// ---- DUTs/AxisControl/ST_AxisControlManualHMI.TcDUT
TYPE ST_AxisControlManualHMI :
STRUCT
	bEnableManualMode							: BOOL;
	bConsequentialError							: BOOL;
	bError										: BOOL;
	nErrorID									: UDINT;
	fSetPos										: LREAL;					// Set position (absolut value from NC)
	fModuloSetPos								: LREAL;					// Actual modulo position (absolut value from NC)
	fSetVelo									: LREAL;					// Set velocity
	fSetTorque									: LREAL;
	fActPos										: LREAL;					// Actual position (absolut value from NC)
	fModuloActPos								: LREAL;					// Actual modulo position (absolut value from NC)
	fActVelo									: LREAL;					// Actual velocity
	fActTorque									: LREAL;
	fPosDiff									: LREAL;					// Position difference (lag distance)
	stCommands									: ST_AxisControlManual;
	stStatus									: REFERENCE TO Tc2_MC2.ST_AxisStatus;
	stParameters								: REFERENCE TO Tc2_MC2.ST_AxisParameterSet;
END_STRUCT
END_TYPE

// ---- DUTs/CapPreScrewer/E_CapPreScrewer.TcDUT

(*
Nazwa:			E_GripperScrewerState
Opis:			Stan zakecarki szczekowej
Wersja:			v0.1
Data:			2023-10-10
Autor:			TW
Urzadzenia:		
Konfiguracja:	
Info:
*)

TYPE E_CapPreScrewer :
(	
	eReady							:= 10,
	ePreparingToPick				:= 20,			
	ePicking						:= 30,
	eVacumCheckPart1				:= 40,
	eVacumCheckPart2				:= 50,
	eVacumCheckPart3				:= 50,
	eVacumCheckPart4				:= 60,
	eTransferingVertical			:= 70,
	eTransferingHorizontal			:= 80,
	eAxisGearIn						:= 82,
	eVerticalDownToCatchPos			:= 90,
	ePositionOverBottle				:= 95,	
	eCatching						:= 100,		
	ePlacing						:= 110,
	eStrawCatcherBack				:= 120,
	eFinding						:= 130,
	eFindingStop					:= 140,
	ePreScrewing					:= 145,
	eScrewing						:= 150,
	eScrewingStop					:= 160,
	eFinished						:= 170,
	eGearOut						:= 175,
	                        		
	eReturning1						:= 180,
	eReturning2						:= 190,
                            		
			                	
	eDone							:= 200,
	eNotDone						:= 300
	


	
):= eReady;
END_TYPE

// ---- DUTs/CapPreScrewer/ST_ADS_Read_Write.TcDUT
TYPE ST_ADS_Read_Write :
STRUCT
	stCtr							: ST_ADS_Write;
	uiHardwerLimitSwitch			: UINT;
END_STRUCT
END_TYPE

// ---- DUTs/CapPreScrewer/ST_ADS_Write.TcDUT
TYPE ST_ADS_Write :
STRUCT
	uiNegativeTorqueLimit	AT %Q* : UINT := 2000;		//10 = 1%
	uiPositiveTorqueLimit	AT %Q* : UINT := 2000;
	siHardwerLimitSwitch		   : SINT;				//Hardwer limit switch: 0 - no limit switch, 1- NC, 1- NO
	
END_STRUCT
END_TYPE

// ---- DUTs/CapPreScrewer/ST_CapPreScrewerCommandsIn.TcDUT
TYPE ST_CapPreScrewerCommandsIn :
STRUCT
	bPendantDownwardMovement		: BOOL;						    // Kaseta sterownicza ruch do góry
	bPendantUpwardMovement			: BOOL; 						// Kaseta sterownicza ruch do dolu
	bPendantUpDownFast				: BOOL;							// Kaseta sterownicza góra/dól- wyższa prędkośc
	bPendantRightwardMovement		: BOOL; 						// Kaseta sterownicza ruch w prawo
	bPendantLeftwardMovement		: BOOL; 						// Kaseta sterownicza ruch w lewo
	bPendantRightLeftFast			: BOOL;							// Kaseta sterownicza lewo/prawo- wyższa prędkośc	
	bChoseRecipe					: BOOL;
	
END_STRUCT
END_TYPE

// ---- DUTs/CapPreScrewer/ST_CapPreScrewerParameters.TcDUT
TYPE ST_CapPreScrewerParameters :
STRUCT
	lrTopZPosition						: LREAL;		//Pozycja bezpieczna załapywarki na osi pionowej
	lrPickZPosition						: LREAL;		//Wysokość pobierania
	lrPickYPosition						: LREAL;		//Pozycja osi poziomej do pobierania
	lrPlaceZPosition					: LREAL;		//Wysokość odkładania - koniec załapywania gwintu
	lrPlaceYPosition					: LREAL;		//Pozycja osi poziomej do odkładania
	lrCartesianCatchZPosition			: LREAL;		//Wysokość osi Z dla zamykania łapacza słomek
	lrCapCatcherZPosition				: LREAL;		//Wysokość zamykaniałapek zakrętek
	lrStrawCatcherZPosition				: LREAL;		//Wysokość otwierania łapaczy słomek
	LrCheckStrawCatcherActuatorZPosition: LREAL;		//
	lrScrewerStartZPosition				: LREAL;		//Wysokość początku zakręcania
	lrGripperOpenPosition				: LREAL;		//Wysokość otwierania chwytaka szyjki butelki
	lrCapCapCatcherRelese				: LREAL;		//Wysokość otwierania chwytaka nakrętki
	lrCatcherTopPosition				: LREAL;		//Pozycja górna osi łapaczy słomek
	lrCatcherCatchingPosition			: LREAL;		//Pozycja łapania słomki
	lrCatcherPlacePosition				: LREAL;		//Pozycja dolna łapacza słomki
	lrCatcherSpeed						: LREAL;		//Prędkość 
	lrCatcherAcceleration				: LREAL;		//Przyspieszenie 
	lrCatcherJerk						: LREAL;		//Zryw 
	lrPickerSpeed						: LREAL;		//Prędkość 
	lrPickerSpeedWhenScrewer			: LREAL;		//Prędkość osi Z przy zakręcaniu
	lrPickerAcceleration				: LREAL;		//Przyspieszenie 
	lrPickerJerk						: LREAL;		//Zryw 
	lrScrewDistance						: LREAL;		//Kąt zakręcania
	lrScrewFinding						: LREAL;		//Kąt szukania gwintu
	lrScrewSpeed						: LREAL;		//Prędkość zakręcania
	lrScrewAcceleration					: LREAL;		//Przyspieszenie
	lrScrewJerk							: LREAL;		//Zryw
	lrBendingDistance					: LREAL;		//Odległość zaokrąglania ruchów manipulatora
	lrStrawInsertDistance				: LREAL;		//Odległość wspulnego ruchu osi Z i łapacza słomek (prowadzenie słomki) 
	
	lrCatcherMaxHight					: LREAL;		//Wysokość maksymalan łapacza słomek
	lrCatcherMinHight					: LREAL;		//Wysokość minimalan łapacza słomek
	lrCatcherHightSV					: LREAL;		//Nastawa wysokości łapacza słomek
	rCatcherHightOffset					: REAL;			//Pozycja bazowania
	rPulseRatio							: REAL;			//
	
	bPickerActiv						: ARRAY [1..4] OF BOOL;
	tTimeVacuumWatchdog					: TIME;

	lrHeightAdditionalBlow				: LREAL;		//Wysokość aktywacji dodatkowego przedmuchu wszystkich ssawek (od zakończenia nakładania nasadki)
	
	//bPicker2Activ						: BOOL;
	//bPicker3Activ						: BOOL;
	//bPicker4Activ						: BOOL;
	
	tWaitInPlacePos						: TIME;
	
	bStrawCatcherON						: BOOL;			//Aktywacja pracy łapacza słomek
	bRejectON							: BOOL;			//Aktywacja odrzucania nasadek przy nieudanym pobraniu
	bVacuumDeactivate					: BOOL;			//Deaktywować podcisnienie
	
	sADS_NetId							: STRING;		//Adres net id dla komunikacji ADS
	nAxisY_ADS_SlaveAddr				: UINT;			//Adres urzadzenia dla komunikacji ADS
	nAxisZ_ADS_SlaveAddr				: UINT;			//Adres urzadzenia dla komunikacji ADS
	nCatcher_ADS_SlaveAddr				: UINT;			//Adres urzadzenia dla komunikacji ADS
	
	lrBottleHight						: LREAL;		//Wysokość butelki
	lrCapHight							: LREAL;		//Wysokość zamknięcia
	lrCapNeckHight						: LREAL;		//Wysokość szyjki zamknięcia
	
END_STRUCT
END_TYPE

// ---- DUTs/CapPreScrewer/ST_FormsCapSorter.TcDUT
TYPE ST_FormsCapSorter :
STRUCT
	bFormPresence 			: BOOL;
	bBottlePresence			: BOOL;
	bFormControlCheck		: BOOL;
	bCapPutDown				: BOOL;
END_STRUCT
END_TYPE

// ---- DUTs/DUTsAdsCommunication/ST_Communication.TcDUT
TYPE ST_Communication :
STRUCT
	
	ePackMLMode						: Tc3_PackML.E_PMLUnitMode;						//Mode 
	ePackMLAutoState				: Tc3_PackML.E_PMLState;							//PackML Auto State
	sPackMLCommand					: ST_PackMLCmdForCom;					//PackML Commands
	
	eError							: S_Error;
	
	bEnable							: BOOL;	
	bCycleStart						: BOOL;
	bCycleStop						: BOOL;
	bCycleReset						: BOOL;
	bManualMode						: BOOL;
	bHoming							: BOOL;
	bHomingDone						: BOOL;	
	bConfectionEnding				: BOOL;
	tCycleTime						: TIME;
	iWatchdog						: INT;
	
	sRecipeName						: STRING(255);							
	sRecipeIndex					: STRING(255);
	
	eMachinePermissions				: ST_MachinePermissions;
	eReservedSignals				: ST_ReservedSignals;
END_STRUCT
END_TYPE

// ---- DUTs/DUTsAdsCommunication/ST_MachinePermissions.TcDUT
TYPE ST_MachinePermissions :
STRUCT
	(* REZERWA *)
	bPermission00 : BOOL;
	(* REZERWA *)
	bPermission01 : BOOL;
	(* REZERWA *)
	bPermission02 : BOOL;
	(* REZERWA *)
	bPermission03 : BOOL;
	(* REZERWA *)
	bPermission04 : BOOL;
	(* REZERWA *)
	bPermission05 : BOOL;
	(* REZERWA *)
	bPermission06 : BOOL;
	(* REZERWA *)
	bPermission07 : BOOL;
	(* REZERWA *)
	bPermission10 : BOOL;
	(* REZERWA *)
	bPermission11 : BOOL;
	(* REZERWA *)
	bPermission12 : BOOL;
	(* REZERWA *)
	bPermission13 : BOOL;
	(* REZERWA *)
	bPermission14 : BOOL;
	(* REZERWA *)
	bPermission15 : BOOL;
	(* REZERWA *)
	bPermission16 : BOOL;
	(* REZERWA *)
	bPermission17 : BOOL;
END_STRUCT
END_TYPE

// ---- DUTs/DUTsAdsCommunication/ST_PackMLCmdForCom.TcDUT
TYPE ST_PackMLCmdForCom :
STRUCT
	bStart						: BOOL;
	bHold						: BOOL;
	bUnHold						: BOOL;
	bSuspend					: BOOL;
	bAbort						: BOOL;
	bStop						: BOOL;
	bComplete					: BOOL;
	bClear						: BOOL;
	bReset						: BOOL;
	bStateComplete				: BOOL;	
END_STRUCT
END_TYPE

// ---- DUTs/DUTsAdsCommunication/ST_ReservedSignals.TcDUT
TYPE ST_ReservedSignals :
STRUCT
	(* REZERWA *)
	bReserved00 : BOOL;
	(* REZERWA *)
	bReserved01 : BOOL;
	(* REZERWA *)
	bReserved02 : BOOL;
	(* REZERWA *)
	bReserved03 : BOOL;
	(* REZERWA *)
	bReserved04 : BOOL;
	(* REZERWA *)
	bReserved05 : BOOL;
	(* REZERWA *)
	bReserved06 : BOOL;
	(* REZERWA *)
	bReserved07 : BOOL;
	(* REZERWA *)
	bReserved10 : BOOL;
	(* REZERWA *)
	bReserved11 : BOOL;
	(* REZERWA *)
	bReserved12 : BOOL;
	(* REZERWA *)
	bReserved13 : BOOL;
	(* REZERWA *)
	bReserved14 : BOOL;
	(* REZERWA *)
	bReserved15 : BOOL;
	(* REZERWA *)
	bReserved16 : BOOL;
	(* REZERWA *)
	bReserved17 : BOOL;
	(* REZERWA *)
	iReserved20 : INT;
	(* REZERWA *)
	iReserved30 : INT;
END_STRUCT
END_TYPE

// ---- DUTs/DUTsAxisOnline/FBsIO/ST_FBGetDriveRefIO.TcDUT
//==================================================================================================
//							Beckhoff Automation Poland
//									18.04.2018
//	Struktura zawierajaca I/O odpowiedniego bloku
//  v1.0	|| TC v 3.1.4022.16		|| - pierwsza wersja
//==================================================================================================
TYPE ST_FBGetDriveRefIO:
STRUCT
	bExecute						: BOOL;								// Rising edge executes cmd
	bBusy							: BOOL;								// Read/Write busy
	bError							: BOOL;								// Read/Write error
	udiErrorID						: UDINT;							// Read/Write error ID
END_STRUCT
END_TYPE

// ---- DUTs/DUTsAxisOnline/FBsIO/ST_FBHoldingBrakeCtrlIO.TcDUT
//==================================================================================================
//							Beckhoff Automation Poland
//									18.05.2018
//	Struktura zawierajaca I/O odpowiedniego bloku
//  v1.0	|| TC v 3.1.4022.16		|| - pierwsza wersja
//==================================================================================================
TYPE ST_FBHoldingBrakeCtrlIO:
STRUCT
	bForceLock 						: BOOL;								// 
	bForceUnlock					: BOOL;								// 
	bBusy							: BOOL;
	bError							: BOOL; 							// General error: parameter or CoE read.
																		// If bError = TRUE and bInitialized = FALSE - error during read motor data.
																		// If bError = TRUE and bInitialized = TRUE and (iAdsErrId <> 0 or iCANopenErrId <> 0) then I2T read error
																		// If bError = TRUE and bInitialized = TRUE and iAdsErrId = 0 and iCANopenErrId = 0 then parameter error: rTorqueLimit outside permitted range rTorqueLimitLow..rTorqueLimitHigh or Empty stDriveRef
	uiAdsErrId						: UINT;								// Forwarded output FB_CoERead_ByDriveRef
	uiSecErrId						: UINT;								// Sercos Error ID for AX5000, CanOpen error ID for AX8000
END_STRUCT
END_TYPE

// ---- DUTs/DUTsAxisOnline/FBsIO/ST_FBMotorMonitoringIO.TcDUT
//==================================================================================================
//							Beckhoff Automation Poland
//									21.05.2018
//	Struktura zawierajaca I/O odpowiedniego bloku
//  v1.0	|| TC v 3.1.4022.16		|| - pierwsza wersja
//==================================================================================================
TYPE ST_FBMotorMonitoringIO:
STRUCT
	bReset							: BOOL;								// Reset FB
	rTorqueLimit					: REAL		:=	500; 				// Bipolar torque limit: 0-500%, resolution 0.1%, value goes to: 16#6072 (Ch A)/ 16#6872 (Ch B)

	bError							: BOOL; 							// General error: parameter or CoE read.
																		// If bError = TRUE and bInitialized = FALSE - error during read motor data.
																		// If bError = TRUE and bInitialized = TRUE and (iAdsErrId <> 0 or iCANopenErrId <> 0) then I2T read error
																		// If bError = TRUE and bInitialized = TRUE and iAdsErrId = 0 and iCANopenErrId = 0 then parameter error: rTorqueLimit outside permitted range rTorqueLimitLow..rTorqueLimitHigh or Empty stDriveRef
	uiAdsErrId						: UINT;								// Forwarded output FB_CoERead_ByDriveRef
	uiSecErrId						: UINT;								// Sercos Error ID for AX5000, CanOpen error ID for AX8000
	bInitialized					: BOOL;								// TRUE - Motor data read without errors, so it's possible to calculate torqe and current values in metric units
	bWarning						: BOOL;								// rCurrentF > rWarningCurrent, be aware to be over permitted range
	rWarningCurrent					: REAL; 							// Continuous Stall Current - motor parameter: 16#6075 (Ch A)/ 16#6875 (Ch B); scalled: [A]
	rTorquePerc						: REAL;								// [%]
	rTorquePercMax					: REAL;								// Max [%]
	rTorque							: REAL; 							// [Nm]
	rTorqueF						: REAL;								// Filtered [Nm]
	rTorqueMax						: REAL;								// Max [Nm]
	rCurrent						: REAL; 							// [A]
	rCurrentF						: REAL;								// Filtered [A]
	rCurrentMax						: REAL;								// Max [A]
	rI2T							: REAL; 							// Thermal Motor Utilization: 16#32C1:02 (Ch A)/ 16#36C1:02 (Ch B); units: [%]
	rI2TMax							: REAL; 							// Max % Nominal
END_STRUCT
END_TYPE

// ---- DUTs/DUTsAxisOnline/FBsIO/ST_FBNcSWLimitSwitchCtrlIO.TcDUT
//==================================================================================================
//							Beckhoff Automation Poland
//									18.04.2018
//	Struktura zawierajaca I/O odpowiedniego bloku
//  v1.0	|| TC v 3.1.4022.16		|| - pierwsza wersja
//==================================================================================================
TYPE ST_FBNcSWLimitSwitchCtrlIO:
STRUCT
	bRead							: BOOL;								// Read SW limit switches values and states
	bWrite							: BOOL;								// Write SW limit switches values and states
	bReset							: BOOL; 							// Not yet
// Set values
	lrSetMinPos						: LREAL;							// SW limit switch minimum
	lrSetMaxPos						: LREAL;							// SW limit switch maximum
	bSetMinMon						: BOOL;								// Enable SW limit switch minimum monitoring
	bSetMaxMon						: BOOL;								// Enable SW limit switch maximum monitoring
// Actual values	
	lrActMinPos						: LREAL;							// Actual SW limit switch minimum
	lrActMaxPos						: LREAL;							// Actual SW limit switch maximum
	bActMinMon						: BOOL;								// SW limit switch minimum monitoring state
	bActMaxMon						: BOOL;								// SW limit switch maximum monitoring stateEND_STRUCT
//	
	bBusy							: BOOL;								// Read/Write busy
	bError							: BOOL;								// Read/Write error
	udiErrorID						: UDINT;							// Read/Write error ID
END_STRUCT
END_TYPE

// ---- DUTs/DUTsAxisOnline/FBsIO/ST_FBReadChannelErrorCodeIO.TcDUT
//==================================================================================================
//							Beckhoff Automation Poland
//									18.04.2018
//	Struktura zawierajaca I/O odpowiedniego bloku
//  v1.0	|| TC v 3.1.4022.16		|| - pierwsza wersja
//==================================================================================================
TYPE ST_FBReadChannelErrorCodeIO:
STRUCT
	bExecute						: BOOL;								// Rising edge executes cmd
	bBusy							: BOOL;
	bError							: BOOL; 							// General error: parameter or CoE read.
	uiAdsErrId						: UINT;								// Forwarded output FB_CoERead_ByDriveRef
	uiSecErrId						: UINT;								// Sercos Error ID for AX5000, CanOpen error ID for AX8000
	uiChannelErrorCode				: UINT;								// 603F Error code	0x603F (Ch A)/ 0x683F (Ch B) 	UINT16
	{attribute 'displaymode':='hex'}
	uiChannelErrorCodeHex			: UINT;								// 603F Error code	0x603F (Ch A)/ 0x683F (Ch B) 	UINT16
END_STRUCT
END_TYPE

// ---- DUTs/DUTsAxisOnline/FBsIO/ST_FBSetPositionOffsetIO.TcDUT
//==================================================================================================
//							Beckhoff Automation Poland
//									23.05.2018
//	Struktura zawierajaca I/O odpowiedniego bloku
//  v1.1	|| TC v 3.1.4022.16		|| - zmiana nazwy struktury usuniete CoE
//  v1.0	|| TC v 3.1.4022.16		|| - pierwsza wersja
//==================================================================================================
TYPE ST_FBSetPositionOffsetIO:
STRUCT
	bExecute						: BOOL;								// Rising edge executes cmd
	lrPosition						: LREAL;
	bRelative						: BOOL;
	eFeedback						: Tc2_MC2_Drive.E_PositionOffsetFeedback;
	eMemory							: Tc2_MC2_Drive.E_PositionOffsetMemory;
	bBusy							: BOOL;
	bError							: BOOL;
	udiErrorID						: UDINT;
	uiSecErrId						: UINT;								// Sercos Error ID for AX5000, CanOpen error ID for AX8000
END_STRUCT
END_TYPE

// ---- DUTs/DUTsAxisOnline/FBsIO/ST_McAxisOnlineErrorCollection.TcDUT
//==================================================================================================
//							Beckhoff Automation Poland
//									7.12.2018
//	Struktura zawierajaca wszsytkie bbledy AxisOnline
//  v1.1	|| TC v 3.1.4022.27		|| - dodane opisy bledow w formie zmiennych typu string
//  v1.0	|| TC v 3.1.4022.16		|| - pierwsza wersja
//==================================================================================================
TYPE ST_McAxisOnlineErrorCollection :
STRUCT
	// Error Collection
	bError							: BOOL;						// General Error flag - all error, FB, NC, drive, communication...
	bNcError						: BOOL;
	bFBError						: BOOL;						// Mc FB error
	bCommunicationError				: BOOL;						// ADS, CoE (AX8000), SoE (AX5000)...
	bDriveError						: BOOL;
	uiAdsErrorID					: UINT;						// Forwarded output FB_CoERead_ByDriveRef
	uiSecErrorID					: UINT;						// Sercos Error ID for AX5000, CanOpen error ID for AX8000
	udiErrorID						: UDINT;					// Set Position Offset FB error ID
	udiNcErrorID					: UDINT;					// Nc ErrorID
	{attribute 'displaymode':='hex'}
	udiNcErrorIDHex					: UDINT;					// Nc ErrorID
	udiFBErrorID					: UDINT;					// FB ErrorID
	{attribute 'displaymode':='hex'}
	udiFBErrorIDHex					: UDINT;					// FB ErrorID

	uiDriveErrorID					: UINT;						// 603F Error code	0x603F (Ch A)/ 0x683F (Ch B) 	UINT16
	{attribute 'displaymode':='hex'}
	uiDriveErrorIDHex				: UINT;						// 603F Error code	0x603F (Ch A)/ 0x683F (Ch B) 	UINT16
	sNcError						: STRING(255);				// Error description
	sDriveError						: STRING(255);				// Error description
END_STRUCT
END_TYPE

// ---- DUTs/DUTsAxisOnline/FBsIO/ST_McAxisStatus.TcDUT
//==================================================================================================
//							Beckhoff Automation Poland
//									24.04.2018
//	Struktura zawierajaca najwazniejsze statusy osi
//  v1.0	|| TC v 3.1.4022.16		|| - pierwsza wersja
//==================================================================================================
TYPE ST_McAxisStatus :
STRUCT
	stAxisStatus			: Tc2_MC2.ST_AxisStatus;
	sAxisName				: STRING(31);				// 
	dwAxisId				: DWORD;					// Axis ID
	bNcError				: BOOL;						// Nc Eror flag
	udiNcErrorCode			: UDINT;					// Nc axis error code
	{attribute 'displaymode':='hex'}
	udiNcErrorCodeHex		: UDINT;					// Nc axis error code - hex format
	lrActPos				: LREAL;					// Actual position (absolut value from NC)
	lrModuloActPos			: LREAL;					// Actual modulo position (absolut value from NC)
	lrActVelo				: LREAL;					// Actual velocity
	lrActAcc				: LREAL;					// Actual acceleration
	lrActTorque				: LREAL;
	lrSetPos				: LREAL;					// Set position (absolut value from NC)
	lrSetVelo				: LREAL;					// Set velocity
	lrSetAcc				: LREAL;					// Set acceleration
	lrSetTorque				: LREAL;

	lrPosDiff				: LREAL;					// Position difference (lag distance)
	bAxisReady				: BOOL;						// Axis.Status.Operational
	bHomed					: BOOL;
	bCoupled				: BOOL;
	bAcceptBlockedDrive		: BOOL;						// Force move back from limit switch
END_STRUCT
END_TYPE

// ---- DUTs/DUTsAxisOnline/FBsIO/ST_MCHaltIO.TcDUT
//==================================================================================================
//							Beckhoff Automation Poland
//									18.04.2018
//	Struktura zawierajaca I/O odpowiedniego bloku
//  v1.0	|| TC v 3.1.4022.16		|| - pierwsza wersja
//==================================================================================================
TYPE ST_MCHaltIO:
STRUCT
	bExecute						: BOOL;								// Rising edge executes cmd
	lrDeceleration					: LREAL;
	lrJerk							: LREAL;
	eBufferMode						: Tc2_MC2.MC_BufferMode;
	stOptions						: Tc2_MC2.ST_MoveOptions;
	bDone							: BOOL;
	bBusy							: BOOL;
	bActive							: BOOL;
	bCommandAborted					: BOOL;
	bError							: BOOL;
	udiErrorID						: UDINT;
END_STRUCT
END_TYPE

// ---- DUTs/DUTsAxisOnline/FBsIO/ST_MCHomeIO.TcDUT
//==================================================================================================
//							Beckhoff Automation Poland
//									18.04.2018
//	Struktura zawierajaca I/O odpowiedniego bloku
//  v1.0	|| TC v 3.1.4022.16		|| - pierwsza wersja
//==================================================================================================
TYPE ST_MCHomeIO:
STRUCT
	bExecute						: BOOL;								// Rising edge executes cmd
	lrPosition						: LREAL					:= DEFAULT_HOME_POSITION;
	eHomingMode						: Tc2_MC2.MC_HomingMode;
	eBufferMode						: Tc2_MC2.MC_BufferMode;
	stOptions						: Tc2_MC2.ST_HomingOptions;
	bCalibrationCam					: BOOL;
	bDone							: BOOL;
	bBusy							: BOOL;
	bActive							: BOOL;
	bCommandAborted					: BOOL;
	bError							: BOOL;
	udiErrorID						: UDINT;
END_STRUCT
END_TYPE

// ---- DUTs/DUTsAxisOnline/FBsIO/ST_MCJogIO.TcDUT
//==================================================================================================
//							Beckhoff Automation Poland
//									18.04.2018
//	Struktura zawierajaca I/O odpowiedniego bloku
//  v1.0	|| TC v 3.1.4022.16		|| - pierwsza wersja
//==================================================================================================
TYPE ST_MCJogIO:
STRUCT
	bSlowForward					: BOOL;
	bSlowBackward					: BOOL;
	bFastForward					: BOOL;
	bFastBackward					: BOOL;
	bJogForward						: BOOL;
	bJogBackwards					: BOOL;
	eMode							: Tc2_MC2.E_JogMode;
	lrPosition						: LREAL;
	lrVelocity						: LREAL;
	lrAcceleration					: LREAL;
	lrDeceleration					: LREAL;
	lrJerk							: LREAL;
	bDone							: BOOL;
	bBusy							: BOOL;
	bActive							: BOOL;
	bCommandAborted					: BOOL;
	bError							: BOOL;
	udiErrorID						: UDINT;
END_STRUCT
END_TYPE

// ---- DUTs/DUTsAxisOnline/FBsIO/ST_MCMoveAbsoluteIO.TcDUT
//==================================================================================================
//							Beckhoff Automation Poland
//									18.04.2018
//	Struktura zawierajaca I/O odpowiedniego bloku
//  v1.0	|| TC v 3.1.4022.16		|| - pierwsza wersja
//==================================================================================================
TYPE ST_MCMoveAbsoluteIO:
STRUCT
	bExecute						: BOOL;								// Rising edge executes cmd
	lrPosition						: LREAL;
	lrVelocity						: LREAL;
	lrAcceleration					: LREAL;
	lrDeceleration					: LREAL;
	lrJerk							: LREAL;
	eBufferMode						: Tc2_MC2.MC_BufferMode;
	stOptions						: Tc2_MC2.ST_MoveOptions;
	bDone							: BOOL;
	bBusy							: BOOL;
	bActive							: BOOL;
	bCommandAborted					: BOOL;
	bError							: BOOL;
	udiErrorID						: UDINT;
END_STRUCT
END_TYPE

// ---- DUTs/DUTsAxisOnline/FBsIO/ST_MCMoveModuloIO.TcDUT
//==================================================================================================
//							Beckhoff Automation Poland
//									18.04.2018
//	Struktura zawierajaca I/O odpowiedniego bloku
//  v1.0	|| TC v 3.1.4022.16		|| - pierwsza wersja
//==================================================================================================
TYPE ST_MCMoveModuloIO:
STRUCT
	bExecute						: BOOL;								// Rising edge executes cmd
	lrPosition						: LREAL;
	lrVelocity						: LREAL;
	lrAcceleration					: LREAL;
	lrDeceleration					: LREAL;
	lrJerk							: LREAL;
	eDirection						: Tc2_MC2.MC_Direction 		:= MC_Positive_Direction; // MC_Positive_Direction := 1, MC_Shortest_Way, MC_Negative_Direction, MC_Current_Direction
	eBufferMode						: Tc2_MC2.MC_BufferMode;
	stOptions						: Tc2_MC2.ST_MoveOptions;
	bDone							: BOOL;
	bBusy							: BOOL;
	bActive							: BOOL;
	bCommandAborted					: BOOL;
	bError							: BOOL;
	udiErrorID						: UDINT;
END_STRUCT
END_TYPE

// ---- DUTs/DUTsAxisOnline/FBsIO/ST_MCMoveRelativeIO.TcDUT
//==================================================================================================
//							Beckhoff Automation Poland
//									18.04.2018
//	Struktura zawierajaca I/O odpowiedniego bloku
//  v1.0	|| TC v 3.1.4022.16		|| - pierwsza wersja
//==================================================================================================
TYPE ST_MCMoveRelativeIO:
STRUCT
	bExecute						: BOOL;								// Rising edge executes cmd
	lrDistance						: LREAL;
	lrVelocity						: LREAL;
	lrAcceleration					: LREAL;
	lrDeceleration					: LREAL;
	lrJerk							: LREAL;
	eBufferMode						: Tc2_MC2.MC_BufferMode;
	stOptions						: Tc2_MC2.ST_MoveOptions;
	bDone							: BOOL;
	bBusy							: BOOL;
	bActive							: BOOL;
	bCommandAborted					: BOOL;
	bError							: BOOL;
	udiErrorID						: UDINT;
END_STRUCT
END_TYPE

// ---- DUTs/DUTsAxisOnline/FBsIO/ST_MCMoveVelocityIO.TcDUT
//==================================================================================================
//							Beckhoff Automation Poland
//									18.04.2018
//	Struktura zawierajaca I/O odpowiedniego bloku
//  v1.0	|| TC v 3.1.4022.16		|| - pierwsza wersja
//==================================================================================================
TYPE ST_MCMoveVelocityIO:
STRUCT
	bExecute						: BOOL;								// Rising edge executes cmd
	lrVelocity						: LREAL;
	lrAcceleration					: LREAL;
	lrDeceleration					: LREAL;
	lrJerk							: LREAL;
	eDirection						: Tc2_MC2.MC_Direction 		:= MC_Positive_Direction; // MC_Positive_Direction := 1, MC_Shortest_Way, MC_Negative_Direction, MC_Current_Direction
	eBufferMode						: Tc2_MC2.MC_BufferMode;
	stOptions						: Tc2_MC2.ST_MoveOptions;
	bDone							: BOOL;
	bInVelocity						: BOOL;								// The same meaning as bDone
	bBusy							: BOOL;
	bActive							: BOOL;
	bCommandAborted					: BOOL;
	bError							: BOOL;
	udiErrorID						: UDINT;
END_STRUCT
END_TYPE

// ---- DUTs/DUTsAxisOnline/FBsIO/ST_MCPowerIO.TcDUT
//==================================================================================================
//							Beckhoff Automation Poland
//									18.04.2018
//	Struktura zawierajaca I/O odpowiedniego bloku
//  v1.0	|| TC v 3.1.4022.16		|| - pierwsza wersja
//==================================================================================================
TYPE ST_MCPowerIO:
STRUCT
	bEnable							: BOOL;
	bEnable_Positive				: BOOL;
	bEnable_Negative				: BOOL;
	lrOverride						: LREAL := 100.0;
	eBufferMode						: Tc2_MC2.MC_BufferMode;
	stOptions						: Tc2_MC2.ST_PowerOptions;
	bStatus							: bool; // Same meaning as Done
	bBusy							: BOOL;
	bActive							: BOOL;
	bError							: BOOL;
	udiErrorID						: UDINT;
END_STRUCT
END_TYPE

// ---- DUTs/DUTsAxisOnline/FBsIO/ST_MCReadDriveAddressIO.TcDUT
//==================================================================================================
//							Beckhoff Automation Poland
//									18.04.2018
//	Struktura zawierajaca I/O odpowiedniego bloku
//  v1.0	|| TC v 3.1.4022.16		|| - pierwsza wersja
//==================================================================================================
TYPE ST_MCReadDriveAddressIO:
STRUCT
	bExecute						: BOOL;								// Rising edge executes cmd
	bDone							: BOOL;
	bBusy							: BOOL;
	bError							: BOOL;
	udiErrorID						: UDINT;
END_STRUCT
END_TYPE

// ---- DUTs/DUTsAxisOnline/FBsIO/ST_MCReadParameterSetIO.TcDUT
//==================================================================================================
//							Beckhoff Automation Poland
//									18.04.2018
//	Struktura zawierajaca I/O odpowiedniego bloku
//  v1.0	|| TC v 3.1.4022.16		|| - pierwsza wersja
//==================================================================================================
TYPE ST_MCReadParameterSetIO :
STRUCT
	bExecute						: BOOL;								// Rising edge executes cmd
	bDone							: BOOL;
	bBusy							: BOOL;
	bError							: BOOL;
	udiErrorID						: UDINT;
END_STRUCT
END_TYPE

// ---- DUTs/DUTsAxisOnline/FBsIO/ST_MCResetIO.TcDUT
//==================================================================================================
//							Beckhoff Automation Poland
//									18.04.2018
//	Struktura zawierajaca I/O odpowiedniego bloku
//  v1.0	|| TC v 3.1.4022.16		|| - pierwsza wersja
//==================================================================================================
TYPE ST_MCResetIO:
STRUCT
	bExecute						: BOOL;								// Rising edge executes cmd
	bDone							: BOOL;
	bBusy							: BOOL;
	bError							: BOOL;
	udiErrorID						: UDINT;
END_STRUCT
END_TYPE

// ---- DUTs/DUTsAxisOnline/FBsIO/ST_MCSetPositionIO.TcDUT
//==================================================================================================
//							Beckhoff Automation Poland
//									18.04.2018
//	Struktura zawierajaca I/O odpowiedniego bloku
//  v1.0	|| TC v 3.1.4022.16		|| - pierwsza wersja
//==================================================================================================
TYPE ST_MCSetPositionIO:
STRUCT
	bExecute						: BOOL;								// Rising edge executes cmd
	lrPosition						: LREAL;
	bMode							: BOOL;								// RELATIVE = True, ABSOLUTE = False (Default)
	stOptions						: Tc2_MC2.ST_SetPositionOptions;
	bDone							: BOOL;
	bBusy							: BOOL;
	bError							: BOOL;
	udiErrorID						: UDINT;
END_STRUCT
END_TYPE

// ---- DUTs/DUTsAxisOnline/FBsIO/ST_MCStopIO.TcDUT
//==================================================================================================
//							Beckhoff Automation Poland
//									18.04.2018
//	Struktura zawierajaca I/O odpowiedniego bloku
//  v1.0	|| TC v 3.1.4022.16		|| - pierwsza wersja
//==================================================================================================
TYPE ST_MCStopIO:
STRUCT
	bExecute						: BOOL;								// Rising edge executes cmd
	lrDeceleration					: LREAL; 
	lrJerk							: LREAL;
	stOptions						: Tc2_MC2.ST_MoveOptions;
	bDone							: BOOL;
	bBusy							: BOOL;
	bActive							: BOOL;
	bCommandAborted					: BOOL;
	bError							: BOOL;
	udiErrorID						: UDINT;
END_STRUCT
END_TYPE

// ---- DUTs/DUTsAxisOnline/ST_AX5000Diag.TcDUT
TYPE ST_AX5000Diag :
STRUCT
(* NC-Status *)
	nNCAxisID							: UDINT;
	bOperational						: BOOL;
	bC1DError							: BOOL;
	bWcStateError						: BOOL;
	bAxisError							: BOOL;
	iAxisErrorCode						: UDINT;

(* Drive Diag *)
	strDriveType						: STRING(19);
	strMotorType						: STRING(31);
	wDriveStatus						: WORD;
	wClass1Diag							: WORD;
	stClass1Diag						: ST_AX5000_C1D;
	stDriveStatus						: ST_AX5000DriveStatus;
	stEcSlaveStateBits					: ST_EcSlaveStateBits;
	stEcSlaveState						: ST_EcSlaveState;
	bPreopToSafeOpError					: BOOL;
	bSafeOpToOpError					: BOOL;
	stCPxInvParamList					: ST_SoE_CPxInvParamList;
	iDiagNumber							: UDINT;
	stDiagNumberList					: ST_SoE_DiagNumList;
	strDiagMessage						: STRING;
END_STRUCT
END_TYPE

// ---- DUTs/DUTsAxisOnline/ST_McAxisOnline.TcDUT
//==================================================================================================
//							Beckhoff Automation Poland
//									18.05.2018
//	Struktura interfejsu do obslugi Axis Online
//	v1.1	|| TC v 3.1.4022.16		|| - zmiana nazw struktur 
// 									 ST_FBCoEAX8000SetPositionOffsetIO 	--> ST_FBCoESetPositionOffsetIO
// 									 ST_FBHoldingBrakeCtrlAX8000IO 		--> ST_FBHoldingBrakeCtrlIO
// 									 ST_FBMotorMonitoringAX8000IO 		--> ST_FBMotorMonitoringIO
//  v1.0	|| TC v 3.1.4022.16		|| - pierwsza wersja
//==================================================================================================
TYPE ST_McAxisOnline :
STRUCT
	// Base administration
	mcPower							: ST_MCPowerIO;
	mcStop							: ST_MCStopIO;
	mcHalt							: ST_MCHaltIO;
	mcSS1							: ST_MCStopIO;
	mcSS2							: ST_MCStopIO;
	mcReset							: ST_MCResetIO;
	mcHome							: ST_MCHomeIO;
	mcSetPosition					: ST_MCSetPositionIO;
	stSetPositionOffset				: ST_FBSetPositionOffsetIO;
	// Base move
	mcMoveAbsolute					: ST_MCMoveAbsoluteIO;
	mcMoveRelative					: ST_MCMoveRelativeIO;
	mcMoveVelocity					: ST_MCMoveVelocityIO;
	mcMoveModulo					: ST_MCMoveModuloIO;
	mcMoveAbsolute2					: ST_MCMoveAbsoluteIO;
	mcMoveRelative2					: ST_MCMoveRelativeIO;
	mcMoveVelocity2					: ST_MCMoveVelocityIO;
	mcMoveModulo2					: ST_MCMoveModuloIO;
	mcJog							: ST_MCJogIO;
	// States, parameters, monitoring and diag
	stMotorMonitoring				: ST_FBMotorMonitoringIO;
	stHoldingBrake					: ST_FBHoldingBrakeCtrlIO;
	stNcLimitSwitch					: ST_FBNcSWLimitSwitchCtrlIO;
	stAxisParameter					: Tc2_MC2.ST_AxisParameterSet;
	stDriveRef						: Tc2_EtherCAT.ST_DriveRef;
	stDriveAddress					: Tc2_MC2.ST_DriveAddress;
	stChannelErrorCode				: ST_FBReadChannelErrorCodeIO;
	stStatus						: ST_McAxisStatus;
	// FBs
	stGetDriveRef					: ST_FBGetDriveRefIO;					// IO for FB_GetDriveRef
	mcReadDriveAddress				: ST_MCReadDriveAddressIO;				// IO for MC_ReadDriveAddress
	mcReadParameterSet				: ST_MCReadParameterSetIO;				// IO for MC_ReadParameterSet
	stError							: ST_McAxisOnlineErrorCollection;		// Error collection for all Axis Online functions
	bError							: BOOL;									// General Error flag - all error, FB, NC, drive, communication... check stError for detail
END_STRUCT
END_TYPE

// ---- DUTs/DUTsDiagnostics/E_DiagState.TcDUT
{attribute 'qualified_only'}
{attribute 'strict'}
TYPE E_DiagState :
(
	eOK						:= 10,
	eError					:= 20,
	eResetting				:= 30
);
END_TYPE

// ---- DUTs/DUTsDiagnostics/ST_FrmWcDiag.TcDUT
TYPE ST_FrmWcDiag :
STRUCT
	iNum					:DINT;
	sBin					:String;
END_STRUCT
END_TYPE

// ---- DUTs/DUTsNew/E_Actuator.TcDUT
{attribute 'qualified_only'}
{attribute 'strict'}
TYPE E_Actuator :
(
	eDisabled					:= 0,					// Stan nieaktywnosci             	
	eAborted                    := 1,                   // Stan bezpiecznego zatrzymania  
	eAborting                   := 2,                   // Stan bezpiecznego zatrzymywania
	eError                      := 3,                   // Stan bledu 				                                
	ePreparingToReady           := 7,                   // Stan przygotowywania do gotowosci           
	ePreparingToDisable         := 8,                   // Stan przygotowywania do nieaktywnosci                               
	eReady                      := 10,					// Stan gotowosci
	eResetting					:= 13,					// Stan resetowania bledu
	eRunningToPosition1			:= 15,       
	eRunningToPosition2			:= 16,                                          
	eRunning					:= 98,	                // Stan wykonywania ruchu 
    eNotdone                    := 99,	                // Stan niezakonczenia wykonywanego	                                     
    eDone                       := 100,                  // Stan zakonczenia wykonywanego ruchu   
	eDoneToPosition1            := 101,                  // Stan zakonczenia wykonywanego ruchu 
	eDoneToPosition2            := 102                  // Stan zakonczenia wykonywanego ruchu  
);
END_TYPE

// ---- DUTs/DUTsNew/E_Barrier.TcDUT
{attribute 'qualified_only'}
{attribute 'strict'}
TYPE E_Barrier :
(
	eDisabled 			:= 0,	
	eError				:= 1,				// Stan nieaktywnosci (Stacja wyłączona)             
	eReady				:= 2,				// Stan gotowści do ruchu
	eWaitingToClose		:= 20,				// Stan oczekiwania na zamknięcie ( 1 faza, 4 wagi)
	eWaitingToOpen		:= 21,				// Stan oczekiwania na otwaricie ( 1 faza, 2 wagi)
	eClose				:= 30,				// Stan zamykania
	eOpen				:= 40,				// Stan otwarcia
	eDone				:= 50				// Wykonano cykl 
):=eDisabled;
END_TYPE

// ---- DUTs/DUTsNew/E_WeightLiftStationState.TcDUT
TYPE E_WeightLiftStationState :
(
	eDisabled					:= 0,			//Stan wyłączony
	eReady						:= 10,			//Sprawdzam co się dzieje ze stacją
	ePrepareToStorageOfForms	:= 20,			//Przygotowywanie do magazynowania formatek
	eStorageOfForms				:= 30,			//Magazynuje formatki oraz podnoszę wagę
	eWeighingCycleStart			:= 40,			//Rozpoczęcie Ważenie
	eWeighingCycleON			:= 50,			//Ważenie
	eWeightLiftDown				:= 60,			//Opuszczanie formatek
	eDepartureOfForms			:= 70,			//Wypuszczamy formatki
	eDone						:= 80,			//Cykl skończony
	eRepair						:= 90			//Naprawa stacji
);
END_TYPE

// ---- DUTs/DUTsPackMLStateMachine/E_PackMLCommand.TcDUT
{attribute 'qualified_only'}
{attribute 'strict'}
TYPE E_PackMLCommand :
(
	eUndefined 				:= 0,
	eReset					:= 1,
	eStart					:= 2,
	eStop					:= 3,
	eHold					:= 4,
	eUnhold					:= 5,
	eSuspend 				:= 6,
	eUnsuspend				:= 7,
	eAbort 					:= 8,
	eClear					:= 9
	
);
END_TYPE

// ---- DUTs/DUTsPackMLStateMachine/E_PackMLMode.TcDUT
{attribute 'qualified_only'}
TYPE E_PackMLMode : 
(
	eUndefined		:=  0,
	eAutomatic		:=  1,
	eMaintenance 	:=  2,
	eManual 		:=  3
);
END_TYPE

// ---- DUTs/DUTsPackMLStateMachine/E_PackMLState.TcDUT
{attribute 'qualified_only'}
TYPE E_PackMLState : (
(* states according to PackTags v3.0 *)
	eUndefined				:=  0, //----Nieużywany
	eClearing 				:=  1, //----Nieużywany
	eStopped 				:=  2, //Błąd
	eStarting 				:=  3, //Uruchamianie
	eIdle 					:=  4, //Postój
	eSuspended 				:=  5, //---Nieużywany
	eExecute 				:=  6, //Praca
	eStopping	 			:=  7, //Zatrzymywanie
	eAborting 				:=  8, //Zatrzymywanie awaryjne
	eAborted 				:=  9, //Zatrzymano awaryjnie
	eHolding 				:= 10, //---Nieużywany
	eHeld 					:= 11, //---Nieużywany
	eUnholding 				:= 12, //---Nieużywany
	eSuspending 			:= 13, //---Nieużywany
	eUnsuspending 			:= 14, //---Nieużywany
	eResetting 				:= 15, //Resetowanie błędu, bazowanie
	eCompleting 			:= 16, //---Nieużywany
	eComplete	 			:= 17  //---Nieużywany
);
END_TYPE

// ---- DUTs/E_BottleFeederState.TcDUT
(*
Nazwa:			E_BottleFeederState
Opis:			Stan podajnika butlek
Wersja:			v0.1
Data:			2022-04-11
Autor:			DJ
Urzadzenia:		
Konfiguracja:	
Info:
*)
TYPE E_BottleFeederState :
(
	eDisabled					:= 0,  			// Wyłączona
	eError						:= 1, 			// Błąd 
	eReady						:= 2,			// Gotowość
	Homing						:= 3,    		// Bazowanie stacji 
	eHomingDone					:= 4,			// Bazowanie zakończone
	eManualMovements			:= 5,			// Tryb ręczny 
	ePreparingToMove			:= 60,			// Przygotowanie do ruchu
	eCloseFirstGate				:= 70,			// Zamknięcie pierwszego szlabanu
	eMoveToCatch				:= 80,			// Ruch do pobrania
	eCloseGripper				:= 90,			// Zamknięcie chwytaka
	eOpenSecondGate				:= 100,			// Otwarcie drugiego szlabanu
	eGoAbove					:= 110,			// Ruch nad formatkę
	eCloseSecondGate			:= 120,			// Zamknięcie drugiego szlabanu i otwarcie pierwszego
	eCloseStoper				:= 130, 			// Uruchomienie docisku
	eInsterting					:= 140,			// Wkładanie butelki
	eOpenGripper				:= 150,			// Otwieranie chwytaka
	eBackToPosition				:= 160,			// Powrót do pozycji wyjściowej
	eRelaseStoper				:= 170			// Wypuszczanie formatki 
);

END_TYPE

// ---- DUTs/E_CapFeederState.TcDUT
(*
Nazwa:			E_CapFeederState
Opis:			Stany sortera nasadek
Wersja:			v0.1
Data:			2018-10-10
Autor:			DP
Urzadzenia:		
Konfiguracja:	
Info:
*)


TYPE E_CapFeederState :
(
	eDisabled:=0,  		//Wyłączona
	eError:=1,			//Błąd
	eManualMovement:=2, //Tryb serwisowy
	eHoming:=3,			//Bazowanie
	eHomingDone:=4, 	//Koniec bazowania
	eReady:=5,			//Gotowość
	eSleeveLowLevel:=6, //Praca, Niski poziom
	eSorting:=7,		//Praca
	eSleeveFull:=8,		//Zapełniona
	ePreparingToDisable:=10 (*NOWY*) //Przygotowanie do wyłączenia
):=eDisabled;
END_TYPE

// ---- DUTs/E_CapFeederState_1.TcDUT
(*
Nazwa:			E_CapFeederState
Opis:			Stany sortera nasadek
Wersja:			v0.1
Data:			2022-07-13
Autor:			DP
Urzadzenia:		
Konfiguracja:	
Info:
*)


TYPE E_CapFeederState_1 :
(
	eDisabled:=0,			//Wyłączony
	eReady:=1,				//Gotowość
	eSleeveLowLevel:=2, 	//Praca, Niski poziom
	eSorting:=3,			//Praca
	eSleeveFull:=4			//Zapełniona
):=eDisabled;
END_TYPE

// ---- DUTs/E_CapPushingState.TcDUT
(*
Nazwa:			E_LidSealingState
Opis:			Stan wbijania nasadek
Wersja:			v0.1
Data:			2018-10-10
Autor:			TW
Urzadzenia:		
Konfiguracja:	
Info:
*)

TYPE E_CapPushingState :
(               	
	eReady:=1,				//Gotowość
	ePushing:=2,			//Wbijanie
	eHolding:=3,			//Przytrzymywanie
	ePushed:=4,				//Wbito
	eGoingUp:=5			//Podnoszenie
);
END_TYPE

// ---- DUTs/E_CatchStationState.TcDUT
(*
Nazwa:			E_CatchStationState
Opis:			Stany chwytaka
Wersja:			v0.2
Data:			2018-10-18
Autor:			TW
Urzadzenia:		
Konfiguracja:	
Info:
-nowy stan
*)

TYPE E_CatchStationState :
(
	eDisabled:=0,  			//Wyłączona
	eError:=1,				//Błąd
	eManualMovement:=2,		//Tryb serwisowy
	eHoming:=4,				//Bazowanie
	eHomingDone:=5,			//Koniec bazowania
	eReady:=6,				//Gotowość
	eCatching:=7, 			//Chwytanie
	eCatched:=8,  			//Chwycono
	ePreparingToDisable:=9, (*NOWY*) //Przygotowanie do wyłączenia
	eNotCatched:=10       //NIe złapało
):=eDisabled;
END_TYPE

// ---- DUTs/E_CheckerState.TcDUT
(*
Nazwa:			E_CheckerState
Opis:			Stan sprawdzania butelek
Wersja:			v0.3
Data:			2023-05-30
Autor:			DP
Urzadzenia:		
Konfiguracja:	
Info:

*)

TYPE E_CheckerState :
(
	eDisabled:=0,			//Wyłączona
	eError:=1,				//Błąd
	eManualMovement:=2,		//Tryb serwisowy
	eHoming:=3,				//Bazowanie
	eHomingDone:=4,			//Koniec bazowania
	eReady:=5,				//Gotowość
	eFormPresent:=6, 		//Formatka
	eBottleOK:=7,	 		//Butelka OK
	eLidOK:=8,		 		//Platynka OK
	eLidNOK:=9,		 		//Platynka NOK	
	eCapOK:=10,		 		//Nasadka OK
	eCapNOK:=11,		 	//Nasadka NOK
	ePreparingToDisable:=12,//Przygotowanie do wyłączenia
	eChecking := 20
):=eDisabled;
END_TYPE

// ---- DUTs/E_ConveyorState.TcDUT
(*
Nazwa:			E_ConveyorState
Opis:			Stan taśmociągu
Wersja:			v0.1
Data:			2018-10-10
Autor:			DP
Urzadzenia:		
Konfiguracja:	
Info:
*)
(*
TYPE E_ConveyorState :
(
	eDisabled:=0,		//Wyłączony
	eError:=1,			//Błąd
	eManualMovement:=2, //Tryb serwisowy
	eHoming:=3,			//Bazowanie
	eHomingDone:=4,		//Koniec bazowania
	eReady:=5,			//Gotowość
	eStopping:=6,	 //Zatrzymywanie
	eStarting:=7, 	//Uruchamianie
	eWorking:=8	  	//Praca
):=eDisabled;
END_TYPE
*)
TYPE E_ConveyorState :
(
	eDisabled := 0,						// Stan nieaktywnosci (Stacja wyłączona)             
	eAborted := 1,                   	// Stan bezpiecznego zatrzymania (po Abortingu) 
	eAborting := 2,                  	// Stan bezpiecznego zatrzymywania (po EStopie)
	eError := 3,                  	 	// Stan błędu 		
	eResetting := 4,					// Stan resetowania bledu (po Errorze)		                
	eManualMovement := 5,     			// Stan ruchów manualnych         
	eHoming := 6,						// Stan bazowania 
	eHomingDone := 7,                   // Stan wykonania bazowania 
	ePreparingToReady := 8,             // Stan przygotowywania do gotowosci (zawsze przed Ready)           
	ePreparingToDisable := 9,           // Stan przygotowywania do nieaktywnosci (po wyłączeniu Enable)                               
	eReady	:= 10,						// Stan gotowosci 
	eStopping := 11,					// Stan zatrzymywania 
	eStarting := 12,                  	// Stan uruchamiania (po Ready)
	eWorking := 13	               		// Stan wykonywania cyklu (po Startingu), w tym stanie osobny 
):=eDisabled;
END_TYPE

// ---- DUTs/E_DispencerLifterState.TcDUT
(*
Nazwa:			E_DispencerState
Opis:			Stan dozowników
Wersja:			v0.1
Data:			2018-10-10
Autor:			TW
Urzadzenia:		
Konfiguracja:	
Info:
*)

TYPE E_DispencerLifterState :
(
	eDisabled:=0,		//Wyłączony
	eError:=1,			//Błąd
	eManualMovement:=2,	//Tryb serwisowy
	eHoming:=3,			//Bazowanie
	eHomingDone:=4,		//Koniec bazowania
	eReady:=5,			//Gotowość
	ePreparingToDose:=6, //Przygotowanie dozy
	eDosingPh1:=7,		 //1 faza dozowania
	eDosingPh2:=8,		 //2 faza dozowania
	eDosingPh3:=9,		 //3 faza dozowania
	eDosingDone:=10,	 //Dozowanie  zakonczone
	eSucking:=11,		 //Pobieranie masy
	eGoingUp:=12,		 //Podnoszenie
	eAborting:=13,		 //Przerywanie
	ePreparingToDisable:=14,//Wylączanie
	ePulling:=15,		//Przeciaganie
(**)eDoseSucking:=16,	// Podsysanie
(**)eDoseSuckingDone:=17 //Koniec podsysania
):=eDisabled;
END_TYPE

// ---- DUTs/E_DispencerState.TcDUT
(*
Nazwa:			E_DispencerState
Opis:			Stan dozowników
Wersja:			v0.1
Data:			2022-03-15
Autor:			DP
Urzadzenia:		
Konfiguracja:	
Info:
- dodane mycie CIP
*)

TYPE E_DispencerState :
(
	eDisabled:=0,		 	//Wyłączony
	eReady:=5,			 	//Gotowość
	ePreparingToDose:=6, 	//Przygotowanie dozy
	eDosingPh1:=7,		 	//1 faza dozowania
	eDosingPh2:=8,		 	//2 faza dozowania
	eDosingPh3:=9,		 	//3 faza dozowania
	eDosingDone:=10,	 	//Dozowanie  zakonczone
	eDoseSucking:=11,	 	//Podsysanie
	eDoseSuckingDone:=12, 	//Koniec podsysania	
	eSucking:=13,		 	//Pobieranie masy
	eGoingUp:=14,		 	//Podnoszenie
	eAborting:=15,		 	//Przerywanie
	ePreparingToDisable:=16,//Wylączanie
	ePulling:=17,			//Przeciaganie
	eCleaningPreparing:=18,	//Mycie | przejazd do pozycji górnej
	eCleaningReady:=19,		//Mycie | pozycja tłoka w górze
	eCleaning:=20,			//Mycie | w trakcie ruchu w dół
	eCleaningDone:=21		//Mycie | pozycja tłoka w dole
):=eDisabled;
END_TYPE

// ---- DUTs/E_DragStationState.TcDUT
(*
Nazwa:			E_DragStationState
Opis:			Stan stacji przeciągania
Wersja:			v0.1
Data:			2021-10-14
Autor:			DJ
Urzadzenia:		
Konfiguracja:	
Info:
*)


TYPE E_DragStationState :
(
	eDisabled					:= 0,  			// Wyłączona
	eReady						:= 2,			// Gotowość
	ePreparingToMove			:= 4,			// Przygotowanie do ruchu
	eLifting					:= 7, 			// Podnoszenie
	ePrepareToDrag				:= 8, 			// Przygotowanie do przeicagana
	eDraging					:= 9,			// Przeciaganie
	eDragingDone				:= 10,			// Kończenie przeciągania
	eEndingOfDrag				:= 11,			// koniec przeciągania, poprawka pozycji
	eEndingOfDragDone			:= 12,			// koniec poprawki
	eLowering					:= 13,			//Opuszczanie 
	eDraged						:= 14,  		//Powrót do bazy, przeciągnięte
	eDragedDone					:= 15
):=eDisabled;

END_TYPE

// ---- DUTs/E_DragStationStatePneum.TcDUT
(*
Nazwa:			E_DragStationState
Opis:			Stan stacji przeciągania pneumatyczengo
Wersja:			v0.2
Data:			2022-05-18
Autor:			DJ
Urzadzenia:		Przeciąganie butelek
Konfiguracja:	
Info:
*)


TYPE E_DragStationStatePneum :
(
	eDisabled					:= 0,  			//Wyłączona
	eReady						:= 2,				//Gotowość
	ePreparingToMove			:= 4,	//Przygotowanie do ruchu
	eLifting					:= 7, 			//Podnoszenie
	ePrepareToDrag				:= 8, 		//Przygotowanie do przeicagana
	eDraging					:= 9,			//Przeciaganie
	eDragingDone				:= 10,
	eEndingOfDrag				:= 11,
	eEndingOfDragDone			:= 12,
	eLowering					:= 13,			//Opuszczanie 
	eDraged						:= 14,  			//Powrót do bazy, przeciągnięte
	eDragedDone					:= 15
):=eDisabled;

END_TYPE

// ---- DUTs/E_EntranceGatesState.TcDUT
(*
Nazwa:			E_EntranceGatesState
Opis:			Stan szlabanów
Wersja:			v0.1
Data:			2018-10-10
Autor:			TW
Urzadzenia:		
Konfiguracja:	
Info:
*)

TYPE E_EntranceGatesState :
(
	eDisabled:=0,					//Wyłączona
	eError:=1,						//Błąd
	eManualMovement:=2,				//Tryb serwisowy
	eHoming:=4,						//Bazowanie
	eHomingDone:=5,					//Koniec bazownia
	eReady:=6,						//Gotowość
	eInsertingTwoForms:=8,			//Wjazd 2 
	eInsertingOneForm:=9,			//Wjazd 1
	eWaitingForRealeseCommand:=11, 	//Czekanie
	eRealeseTwoForms:=12,			//Wyjazd 2
	eRealeseOneForm:=13,			//Wyjazd 1
	eBlocking:=14,					//Blokowanie (**)
	ePulling:=15,					//Przeciąganie (**)
	ePullingDone:=16,				//Wykonano przeciąganie (**)
	ePreparingToReady:=17,			//Przygotowanie do gotowości
	ePreparingToDisable:=18,		//Pryzgotowanie do wyłączenia
	ePullingToMiddle:=19,			//Przeciąganie do środka (**)
	ePullingToMiddleDone:=20,		//Przeciągnięto do środka(**)
	eStayOpen:=21			//Pozstań otwarty
	
):=eDisabled;
END_TYPE

// ---- DUTs/E_FestoEmcsStState.TcDUT
{attribute 'qualified_only'}
{attribute 'strict'}
TYPE E_FestoEmcsStState :
(
	eUnhomed		:=	0,
	eHoming			:=	5,
	eHomingDone		:=	7,
	eUnknown		:=	10,
	eIn				:=	20,
	eOut			:=	30,
	eInter			:=	40,
	eMoveIn			:=	50,
	eSettingIn		:=	55,
	ePlsIn			:=	56,
	eMoveOut		:=	60,
	eSettingOut		:=	65,
	ePlsOut			:=	66,
	eMoveInter		:=	70,
	eSettingInter	:=	75,
	eError			:=	100,
	eResetting		:=	200,
	eEStop			:=	1000						
);
END_TYPE

// ---- DUTs/E_GripperScrewer.TcDUT
(*
Nazwa:			E_GripperScrewerState
Opis:			Stan zakecarki szczekowej
Wersja:			v0.1
Data:			2018-10-10
Autor:			TW
Urzadzenia:		
Konfiguracja:	
Info:
*)

TYPE E_GripperScrewer :
(	
	
	eReady				:= 1,
	eToPushingPosition	:= 2,
	eToScrewingPosition	:= 3,
	ePushed				:= 4,			
	eFindingScrew		:= 5,			
	eScrewing			:= 6,			
	eGoingUp			:= 7,			
	eDone				:= 8,
	eNotDone			:= 9,
	eHolding			:= 10
	
):= eReady;
END_TYPE

// ---- DUTs/E_MachineState.TcDUT
(*
Nazwa:			E_MachineState
Opis:			Stan masyzny
Wersja:			v0.1
Data:			2018-10-10
Autor:			TW,DP
Urzadzenia:		
Konfiguracja:	
Info:
*)

//{attribute 'strict'}
//{attribute 'qualified_only'}
TYPE E_MachineState :
(
	eOn := 0, //Właczono
	ePower := 1, //Zasilanie
	eIdle := 2,	//Inicjacja
	eWaitingForPositioning := 4, //Czekanie na bazowanie
	ePositioning := 5, //Bazowanie
	eReady := 6, //Gotowa
	eServiceMode := 7, //Tryb Serwisowy
	eEnginesOn := 8, //Silniki włączone
	eCycleStarting := 9, //Start cyklu
	eCycleOn := 10, //Praca
	eStopping := 11, //Zatrzymywanie
	eConfectionStart := 12, //Start konfekcji
	eConfectionEnd := 13, //Stop konfekcji
	eHardError := 20, //Bład safety
	eSoftError := 21, //Bład
	eAfterError := 22, //Przywracanie po błedzie
	eReset := 30 //Resetowanie
);
END_TYPE

// ---- DUTs/E_MassHeatingState.TcDUT
(*
Nazwa:			E_MassHeatingState
Opis:			Stan grzania masy
Wersja:			v0.1
Data:			2018-10-10
Autor:			DP
Urzadzenia:		
Konfiguracja:	
Info:
*)

TYPE E_MassHeatingState :
(
	eDisabled:=0,		//Wyłączona
	eHeating:=1,		//Grzanie
	eReady:=2,			//Gotowość
	eCooling:=3			//Chłodzenie
);
END_TYPE

// ---- DUTs/E_PuckInserterState.TcDUT
(*
Nazwa:			E_PuckInserterState
Opis:			Stan podajnika opakowań
Wersja:			v0.1
Data:			2025-02-06
Autor:			DP
Urzadzenia:		
Konfiguracja:	
Info:
*)
TYPE E_PuckInserterState :
(
	eDisabled					:= 0,  			// Wyłączona
	eError						:= 1, 			// Błąd 
	eReady						:= 2,			// Gotowość
	ePreparingToMove			:= 60,			// Przygotowanie do ruchu
	eTurning					:= 70,			// Obrót
	eTurningDone				:= 80,			// Koniec obrotu
	eGoAbove					:= 110,			// Ruch nad formatkę
	eCloseStoper				:= 130, 		// Uruchomienie docisku
	eInsterting					:= 140,			// Wkładanie butelki
	eBackToPosition				:= 160			// Powrót do pozycji wyjściowej

);

END_TYPE

// ---- DUTs/E_RobotMovState.TcDUT
(*
Nazwa:			E_RobotPickAndPlace
Opis:			Stan robota pick-place
Wersja:			v0.1
Data:			2018-10-10
Autor:			TW
Urzadzenia:		
Konfiguracja:	
Info:
*)
TYPE E_RobotMovState :
(
	
	eReadyPlace						:= 0,		// robot w pozycji gotowości
	ePicking						:= 1,  		// pobieranie 
	ePicked							:= 2,
	ePlacing						:= 3,
    ePlaced							:= 4,
	eRejecting						:= 5,
	eRejected 						:= 6,
	eMovingInkJetStartPositon		:= 7,
	eMovedInkJetStartPositon		:= 8,
	eMovingInkJetStopPositon		:= 9,
	eMovedInkJetStopPositon			:= 10,
	eAborting						:= 11,
	eReturnToReadyPlace				:= 12,
	ePickingAfterEStop				:= 13,
	eMovingWeightPosition			:= 14,
	eMovedWeightPosition			:= 15,
	eMovingAfterWeightPosition		:= 16,
	eMovedAfterWeightPosition		:= 17,
	eMovingRotatedToPlace			:= 18,
	eMovedRoatedToPlace				:= 19
	
);
END_TYPE

// ---- DUTs/E_RollerScrewer.TcDUT
(*
Nazwa:			E_RollerScrewerState
Opis:			Stan zakręcarki rolkowej
Wersja:			v0.1
Data:			2018-10-10
Autor:			DP
Urzadzenia:		
Konfiguracja:	
Info:
*)
TYPE E_RollerScrewer :
(
	eDisabled		:=0,			//Niegotowy
	eReady			:=1,			//Gotowość 
	ePushingCap		:=2,			//Wciskanie
	ePushed			:=4,			//Wciśnięto
	eFindingScrew	:=5,			//Szukanie gwintu
	eScrewing		:=6,			//Zakręcanie
	eGoingUp		:=7,			//Podnoszenie
	eDone			:=8,			//Zakręcono
	eNotDone		:=9,			//Przerywanie
	eHolding		:=10			//Przytrzymywanie

):=eDisabled;
END_TYPE

// ---- DUTs/E_Station.TcDUT
(*
Nazwa:			E_MassHeatingState
Opis:			Stan grzania masy
Wersja:			v0.1
Data:			2018-10-10
Autor:			DP
Urzadzenia:		
Konfiguracja:	
Info:
*)

TYPE E_Station :
(
	eDisabled := 0,						// Stan nieaktywnosci (Stacja wyłączona)             
	eAborted := 1,                   	// Stan bezpiecznego zatrzymania (po Abortingu) 
	eAborting := 2,                  	// Stan bezpiecznego zatrzymywania (po EStopie)
	eError := 3,                  	 	// Stan błędu 		
	eResetting := 4,					// Stan resetowania bledu (po Errorze)		                
	eManualMovement := 5,     			// Stan ruchów manualnych         
	eHoming := 6,						// Stan bazowania 
	eHomingDone := 7,                   // Stan wykonania bazowania 
	ePreparingToReady := 8,             // Stan przygotowywania do gotowosci (zawsze przed Ready)           
	ePreparingToDisable := 9,           // Stan przygotowywania do nieaktywnosci (po wyłączeniu Enable)                               
	eReady	:= 10,						// Stan gotowosci 
	eStopping := 11,					// Stan zatrzymywania 
	eStarting := 12,                  	// Stan uruchamiania (po Ready)
	eRunning := 13,	               		// Stan wykonywania cyklu (po Startingu), w tym stanie osobny 
	eDone	:= 14			// Zakończony cykl running
);
END_TYPE

// ---- DUTs/E_WeightState.TcDUT
(*
Nazwa:			E_WeightState
Opis:			Stan zakręcarki rolkowej
Wersja:			v0.1
Data:			2018-10-10
Autor:			TW
Urzadzenia:		
Konfiguracja:	
Info:
*)
TYPE E_WeightState :
(
	eDisabled:=0,		//Wyłączona
	eReady:=1,	  		//Gotowa
	eWeighting:=2,		//Ważenie
	eWeightingDone:=3	//Koniec ważenia
);
END_TYPE

// ---- DUTs/ServerClientENUMS/E_ConnectionSteps.TcDUT
TYPE E_ConnectionSteps :
(
	eCONNECTION_STATE_IDLE,
	eCONNECTION_STATE_CONNECT_START,
	eCONNECTION_STATE_CONNECT_WAIT,
	eCONNECTION_STATE_DATAEXCHANGE,
	eCONNECTION_STATE_CLOSE_START,
	eCONNECTION_STATE_CLOSE_WAIT,
	eCONNECTION_STATE_ERROR
);
END_TYPE

// ---- DUTs/ServerClientENUMS/E_ServerSteps.TcDUT
TYPE E_ServerSteps :
(
	eSERVER_STATE_IDLE,
	eSERVER_STATE_LISTENER_OPEN_START,
	eSERVER_STATE_LISTENER_OPEN_WAIT,
	eSERVER_STATE_REMOTE_CLIENTS_COMM,
	eSERVER_STATE_REMOTE_CLIENTS_CLOSE,
	eSERVER_STATE_LISTENER_CLOSE_START,
	eSERVER_STATE_LISTENER_CLOSE_WAIT,
	eSERVER_STATE_ERROR
);
END_TYPE

// ---- DUTs/Stations/LidFeeder/E_LidFeederState.TcDUT
(*
Nazwa:			E_LidFeederState
Opis:			Stan zpodajnika platynek
Wersja:			v0.2
Data:			2018-10-18
Autor:			TW
Urzadzenia:		
Konfiguracja:	
Info:
*)

TYPE E_LidFeederState :
(
	eDisabled:=0,	//Wyłączona
	eError:=1,		//Błąd
	eManualMovement:=2,	//Tryb serwisowy
	eHoming:=3,		//Bazowanie
	eHomingDone:=4,	//Koniec bazowania
	eHeaterNotReady:=5,	//Grzanie
	eReady:=6,		//Gotowość
	eSuckingLid:=7,	//Pobieranie
	ePuttingLid:=8,	//Przygotowanie do odlożenia
	ePuttingLid2:=9,	//Nakładanie ostatnie
	eHeating:=10,	//Zgrzewanie
	eLidPutted:=11,	//Odłożona
	eGoingUp:=12,	//Podnoszenie
	ePreparingToDisable:=13 (*NOWY*) //Przygotowanie do wyłączenia
(**)
):=eDisabled;
END_TYPE

// ---- DUTs/Stations/LidSealer/E_LidSealing.TcDUT
(*
Nazwa:			E_LidSealingState
Opis:			Stan zgrzewarki platynek
Wersja:			v0.1
Data:			2018-10-10
Autor:			TW
Urzadzenia:		
Konfiguracja:	
Info:
*)

TYPE E_LidSealing :
(
	eDisabled:=0,		// Wyłączona
	eHeaterNotReady:=1, // Grzanie
	eReady:=2,			// Gotowość
	eSealing:=3,		// Zgrzewanie
	eHeating:=4,		// Grzanie
	eLidSealed:=5,		// Zgrzano
	eGoingUp:=6			// Podnoszenie
):=eDisabled;
END_TYPE

// ---- DUTs/Stations/WickFeeder/E_WickFeederSorterState.TcDUT
(*
Nazwa:			E_CapFeederState
Opis:			Stany sortera nasadek
Wersja:			v0.1
Data:			2018-10-10
Autor:			DP
Urzadzenia:		
Konfiguracja:	
Info:
*)


TYPE E_WickFeederSorterState :
(
	eDisabled:=0,  		//Wyłączona
	eError:=1,			//Błąd
	eManualMovement:=2, //Tryb serwisowy
	eHoming:=3,			//Bazowanie
	eHomingDone:=4, 	//Koniec bazowania
	eReady:=5,			//Gotowość
	eSleeveLowLevel:=6, //Praca, Niski poziom
	eSorting:=7,		//Praca
	eSleeveFull:=8,		//Zapełniona
	ePreparingToDisable:=10 (*NOWY*) //Przygotowanie do wyłączenia
):=eDisabled;
END_TYPE

// ---- DUTs/Stations/WickFeeder/E_WickFeederState.TcDUT
(*
Nazwa:			E_LidFeederState
Opis:			Stan zpodajnika platynek
Wersja:			v0.2
Data:			2018-10-18
Autor:			TW
Urzadzenia:		
Konfiguracja:	
Info:
*)

TYPE E_WickFeederState :
(
	eDisabled:=0,	//Wyłączona
	eError:=1,		//Błąd
	eManualMovement:=2,	//Tryb serwisowy
	eHoming:=3,		//Bazowanie
	eHomingDone:=4,	//Koniec bazowania
	//eHeaterNotReady:=5,	//Grzanie
	eFilling:=5,  //Zapełnianie zasobników
	eReady:=6,		//Gotowość 
	eWickDepotReady:=7,	//Magazynek przed włożeniem
	ePuttingWick:=8,	//Przygotowanie do odlożenia
	//ePuttingLid2:=9,	//Nakładanie ostatnie
	//eHeating:=10,	//Zgrzewanie
	eWickPutted:=11,	//Odłożona
	eGoingUp:=12,	//Podnoszenie
	ePreparingToDisable:=13 (*NOWY*) //Przygotowanie do wyłączenia
(**)
):=eDisabled;
END_TYPE

// ---- DUTs/ST_MoverState.TcDUT
TYPE ST_MoverState :
STRUCT
	bInPlacePosition			: BOOL; 	//Wózek w pozycji wyjmowania zamknięć	
	bPlaceAllowed				: BOOL;		//Zezwolenie na pobranie nasadki
	bInPickPosition				: BOOL; 	//Wózek w pozycjach wkładania zamknięć
	bMovingInPickPos			: BOOL;		//Wózek przemieszcza się w pozycji Pick 
	bWaitingForGoToPickPosition	: BOOL;		//Wózek czeka na przejscie do pick w biezpiecznej pozycji 
	bSlot1InPlacePosition		: BOOL;		//Gniazdo 1 ustawione w pozycji wkładania zamknięć
	bSlot2InPlacePosition		: BOOL;		//Gniazdo 2 ustawione w pozycji wkładania zamknięć
	bSlot3InPlacePosition		: BOOL;		//Gniazdo 3 ustawione w pozycji wkładania zamknięć
	bSlot4InPlacePosition		: BOOL;		//Gniazdo 4 ustawione w pozycji wkładania zamknięć
	stSlotStatus				: ARRAY [1..4] OF ST_SlotStatus;		//Gniazdo zapełnione
	bEmpty						: BOOL;		//Pusty wózek
	bFull						: BOOL; 	//zapełniony wózek
	iSlotNo						: INT;		//Nr gniazda
END_STRUCT
END_TYPE

// ---- DUTs/ST_Point.TcDUT
TYPE ST_Point :
STRUCT
	x : INT;
	y : INT;
END_STRUCT
END_TYPE

// ---- DUTs/ST_Point_1.TcDUT
TYPE ST_Point_1 :
STRUCT
	x : DT;
	y : INT;
END_STRUCT
END_TYPE

// ---- DUTs/ST_SlotStatus.TcDUT
TYPE ST_SlotStatus :
	STRUCT
		bFilled			: BOOL;
		bCupPlaced		: BOOL;
		bTubePresent	: BOOL;
		diPlacedRetry	: DINT;
	END_STRUCT
END_TYPE

// ---- DUTs/S_CycleTimes.TcDUT
(*
Nazwa:			S_CycleTimes
Opis:			Struktura czasów cyklu
Wersja:			v0.1
Data:			2019-08-29
Autor:			DP
Urzadzenia:		
Konfiguracja:	
Info:
*)
TYPE S_CycleTimes :
STRUCT
	bName:STRING; 
	bEnable:BOOL;
	dTime:DINT;
END_STRUCT
END_TYPE

// ---- DUTs/S_Error.TcDUT
(*
Nazwa:			S_Error
Opis:			Struktura bledu
Wersja:			v0.2
Data:			2018-10-10
Autor:			TW
Urzadzenia:		
Konfiguracja:	
Info:
- dodano string2
*)
TYPE S_Error :
STRUCT
	bError				: BOOL; 
	udiStationID		: UDINT;
	sStationName		: STRING;
	nErrorCode			: UDINT;
	sErrorString		: STRING(200);
	sErrorString2		: STRING(200);
	bReset:BOOL;
END_STRUCT
END_TYPE

// ---- DUTs/S_Information.TcDUT
(*
Nazwa:			S_Error
Opis:			Struktura bledu
Wersja:			v0.2
Data:			2018-10-10
Autor:			TW
Urzadzenia:		
Konfiguracja:	
Info:
- dodano string2
*)
TYPE S_Information :
STRUCT 
	udiID				: UDINT;
	wsDescription		: WSTRING;
END_STRUCT
END_TYPE

// ---- DUTs/S_PackageState.TcDUT
(*
Nazwa:			S_PackageState 
Opis:			Struktura formatki
Wersja:			v0.1
Data:			2018-10-10
Autor:			DP
Urzadzenia:		
Konfiguracja:	
Info:
*)
TYPE S_PackageState :
STRUCT
	
	nID									:UDINT;							//Numer butelki
	nCardNumber							:ULINT; 						//Numer karty RFID
	bFormPresent						:BOOL;							//Potwierdzenie obecności formatki na wjeździe karuzeli
	bBottlePresent						:BOOL;							//Potwierdzenie obecności butelki na wjeździe karuzeli
	bDosingTwoPhases					:BOOL;							//Jeżeli wybrano dozowanie dwu fazowe
	nDispencerNr						:INT;							//Numer dozownika który wydozował masę 1-6
	nDispencerNrSecondPhase				:INT;							//Numer dozownika który wydozował masę w drugiej fazie
	tDispencingTime						:TIME;							//Czas dozowania
	tDispencingTimeSecondPhase			:TIME;							//Czas dozowania w drugiej fazie
	lrDoseVolumeSV						:LREAL;							//Zadana wartość dozowania [ml]
	lrDoseVolumeCV						:LREAL;							//Aktualna wydozowana ilość [ml]
	lrDoseVolumeSVSecondPhase			:LREAL;							//Zadana wartość dozowania [ml]
	lrDoseVolumeCVSecondPhase			:LREAL;							//Aktualna wydozowana ilość [ml]
	bDosed								:BOOL;							//Zakońcozno cykl dozowania
	bDoseAborted						:BOOL;							//Przerwano dozowanie
	bDosedSecondPhase					:BOOL;							//Zakońcozno cykl dozowania 2 faz
	bDoseAbortedSecondPhase				:BOOL;							//Przerwano dozowanie 2faz
//	bFormInWheel1						:BOOL;							//Potwierdzenie obecności formatki na 1 wjeździe karuzeli
	bWeighed							:BOOL;							//Zwarzono paczkę
	bWeightAborted						:BOOL;							//Przerwano ważenie
	lrWeightSV							:LREAL;							//Zadana wartość netto [g] 
	lrWeightCV							:LREAL;							//Aktualna wartość netto [g]
	lrWeightMeasuredCV					:LREAL;							//Aktualna wartość odczytana z wagi [g]
	lrMinWeightCV						:LREAL;							//Minimalna waga wartość netto [g]	
	lrMaxWeightCV						:LREAL;							//Maksymalna waga wartość netto [g]		
	lrWeightDif							:LREAL;							//Różnica pomiarów				
	bWeightOK							:BOOL;							//Waga zgodna z zakresem tolerancji
	bWeightTooLow						:BOOL;							//Waga za niska
	bWeightTooHigh						:BOOL;							//Waga za wysoka
	tWeightingTime						:TIME;							//Czas ważenia
	bLidPutted							:BOOL;							//Platynka położona 
	bLidPutAborted						:BOOL;							//Odkładanie platynki wycofane w trakcie odkładania
	tLidPuttingTime						:TIME;							//Czas odkładania platynki
	lrPreSealingTime					:LREAL;							//Czas zgrzewania wstępnego
	lrPreSealingTemp					:LREAL;							//Temperatura zgrzewania wstępnego
	bLidPuttedChecked					:BOOL;							//Platynka sprawdzona 
	bLidPuttedOK						:BOOL;							//Platynka sprawidłowo nałożona
	bLidSealed							:BOOL;							//Platynka zgrzana
	bLidSealingAborted					:BOOL;							//Zgrzanie platynki wycofane
	tLidSealingTime						:TIME;							//Czas zgrzewania platynki
	lrLidSealingTemp					:LREAL;							//Temperatura zgrzewania zasadniczego
	bROPPPutted							:BOOL;							//ROPP nasadka ok
	bROPPPuttedChecked					:BOOL;							//ROPP nasadka sprawdzona
	bROPPCapped							:BOOL;							//ROPP ok
	bROPPCappingAborted					:BOOL;							//ROPP nok
	tROPPCappingTime					:TIME;							//Czas ROPPowania
	bROPPCappingOK						:BOOL;							//ROPP nasadka ok za
	bROPPCappingChecked					:BOOL;							
	bCapSorterPutted					:BOOL;							//Nałozono nakrętke przez sorter
	bCapSorterPuttedAborted				:BOOL;							//Nałozono nakrętke przez sorter	
	tCapSorterPuttingTime				:TIME;							//Czas Nałozono nakrętke przez sorter		
	bCapPutted							:BOOL;							//Nałozono nakrętke
	bCapPuttedNOK						:BOOL;							//Nałozono nakrętke NOK
	bCapChecked							:BOOL;							//Nakrętka sprawdzona
	bCapOK								:BOOL;							//Nakrętka OK
//	bCapPushed							:BOOL;							//Wbito nasadke
//	bCapPushingAborted					:BOOL;							//Przerwano wbijanie
//	tCapPushingTime						:TIME;							//Czas wbijania nasadki
//	bFormInWheel2						:BOOL;							//Potwierdzenie obecności formatki na 2 wjeździe karuzeli
	bCapGripperScrewed					:BOOL;							//Nakrętka zakręcona
	bCapGripperScrewAborted				:BOOL;							//Wycofanie z zakręcania nakrętki
	tCapGripperScrewingTime				:TIME;							//Czas zakręcania
//	bCapRollerScrewed					:BOOL;							//Nakrętka zakręcona
//	bCapRollerScrewAborted				:BOOL;							//Wycofanie z zakręcania nakrętki
//	tCapRollerScrewingTime				:TIME;							//Czas zakręcania
	bCapCorrectPutted					:BOOL;							//Nałozono nakrętke
	bCapCorrectChecked					:BOOL;							//Nakrętka sprawdzona
	bCapCorrectNOK						:BOOL;							//Nakrętka NOT OK
	bCapCorrectCapOn					:BOOL;							//Nakrętka obecna
	
	bCapCorrectCheckCameraOK			:BOOL;							//Nakrętka orientacja OK
	bCapCorrectCheckCameraChecked		:BOOL;							//Nakrętka orientacja sprawdzono
	
	bBottleTransferedToExit				:BOOL;							//Butelka przeniesiona na transporter odrzuconych butelek
	bBottleTransferedToLabeler			:BOOL;							//Butelka przeniesiona na etykieciarkę
	
	bTested								: BOOL;
	bTested2							: BOOL;
	bTested3							: BOOL;
	bTested4							: BOOL;
END_STRUCT
END_TYPE

// ---- DUTs/S_RFIDCheck.TcDUT
(*
Nazwa:			S_RFIDCheck
Opis:			sprawdzanie RFID
Wersja:			v0.1
Data:			2024-12-03
Autor:			
Urzadzenia:		
Konfiguracja:	
Info:

*)
TYPE S_RFIDCheck :
STRUCT 
	iNumber				: INT;		//Numer RFID	
	iReaded1			: INT;		//Odczytano z czytnika nr 1
	iReaded2			: INT;		//Odczytano z czytnika nr 2
	iReaded3			: INT;		//Odczytano z czytnika nr 3
	iReaded4			: INT;		//Odczytano z czytnika nr 4
	iReaded5			: INT;		//Odczytano z czytnika nr 5
END_STRUCT
END_TYPE

// ---- DUTs/S_Warning.TcDUT
(*
Nazwa:			S_Warning 
Opis:			Struktura ostrzezen
Wersja:			v0.1
Data:			2018-10-10
Autor:			DP
Urzadzenia:		
Konfiguracja:	
Info:
*)
TYPE S_Warning :
STRUCT
	bWarning:BOOL; 
	bAcknowledge:BOOL;
	sDescription:STRING;
	udiWarningCode:UDINT;
END_STRUCT
END_TYPE

// ---- POUs/Recipes/NewRecipes/Components/ST_BoolParametr.TcDUT
TYPE ST_BoolParametr :
STRUCT
	bValue												:	BOOL;
	bOldValue											:	BOOL;
	bDefault											:	BOOL;
	wsInfoCaption										:	WSTRING(100);
	wsCaption1											:	WSTRING(50);
	wsCaption2											:	WSTRING(50);
	bUse2caption										:	BOOL;
END_STRUCT
END_TYPE

// ---- POUs/Recipes/NewRecipes/Components/ST_DiParametrr.TcDUT
TYPE ST_DiParametrr :
STRUCT
	diValue											:	DINT;
	diOldValue											:	DINT;
	diMinLimit											:	DINT;
	diMaxLimit											:	DINT;
	diDefault											:	DINT;
	diColor											:	DINT	:=	16#FFFFAF1C;	
	wsInfoCaption										:	WSTRING(100);	
	wsCaption1											:	WSTRING(50);
	wsCaption2											:	WSTRING(50);
	bUse2caption										:	BOOL;
	wsUnit												:	WSTRING;
END_STRUCT
END_TYPE

// ---- POUs/Recipes/NewRecipes/Components/ST_LrParametr.TcDUT
TYPE ST_LrParametr :
STRUCT
	lrValue												:	LREAL;
	lrOldValue											:	LREAL;
	lrMinLimit											:	LREAL;
	lrMaxLimit											:	LREAL;
	lrDefault											:	LREAL;
	wsInfoCaption										:	WSTRING(120);	
	wsCaption1											:	WSTRING;
	wsCaption2											:	WSTRING;
	udiColor											:	UDINT	:=	16#FFF0F0F0;	
	bUse2caption										:	BOOL;
	wsUnit												:	WSTRING;
END_STRUCT
END_TYPE

// ---- POUs/Recipes/NewRecipes/Components/ST_TextListParametr.TcDUT
TYPE ST_TextListParametr :
STRUCT
	aWStringTable : ARRAY [0..3] OF WSTRING := ["Butelka okrągła", "Butelka płaska", "Słoik", "Karton jednostkowy"];
	eArrayNumber										:	E_ProductType;
END_STRUCT
END_TYPE

// ---- POUs/Recipes/NewRecipes/Components/ST_UdiParametr.TcDUT
TYPE ST_UdiParametr :
STRUCT
	udiValue											:	UDINT;
	udiOldValue											:	UDINT;
	udiMinLimit											:	UDINT;
	udiMaxLimit											:	UDINT;
	udiDefault											:	UDINT;
	udiColor											:	UDINT	:=	16#FFFFAF1C;	
	wsInfoCaption										:	WSTRING(100);	
	wsCaption1											:	WSTRING(50);
	wsCaption2											:	WSTRING(50);
	bUse2caption										:	BOOL;
	wsUnit												:	WSTRING;
END_STRUCT
END_TYPE

// ---- POUs/Recipes/NewRecipes/E_MacroProductProcessRegister.TcDUT
{attribute 'qualified_only'}
{attribute 'strict'}
TYPE E_MacroProductProcessRegister :
(
	eUnknown									:=	0,
	
	eEmpting									:=	10,
	eEmpty			 							:= 	20,
	
	ePuttingIn		 							:= 	30,
	eFull										:=	40,
	eNotFull									:=	50
//	ePickingToWait								:=	60,
//	ePickedAndWaiting							:=	70	
);
END_TYPE

// ---- POUs/Recipes/NewRecipes/E_ProductType.TcDUT
{attribute 'qualified_only'}
//{attribute 'strict'}
TYPE E_ProductType :
(

	eRoundBottle	:= 	0,
	eFlatBottle 	:= 	1,
	eJar			:=	2,	
	eCarton			:=	3
);
END_TYPE

// ---- POUs/Recipes/NewRecipes/RecipeList/E_FileOpSteps.TcDUT
{attribute 'qualified_only'}
{attribute 'strict'}
TYPE E_FileOpSteps :
(
	eNop 					:=	0,
	eStartOpen				:=	10,
	eWaitOpen				:=	20,
	eStartOper				:=	30,
	eWaitOper				:=	40,
	eStartClose				:=	50,
	eWaitClose				:=	60
);
END_TYPE

// ---- POUs/Recipes/NewRecipes/RecipeParts/ST_BoxRobotRecipe.TcDUT
TYPE ST_BoxRobotRecipe :
STRUCT
	wsCaption											:	WSTRING;	//Nazwa stacji	

	stPickOffsetX									:	ST_LrParametr;	//	Offset poz pobierania x 1mm
	stPickOffsetY									:	ST_LrParametr;	//	Offset poz pobierania x 1mm
	stPickOffsetZ									:	ST_LrParametr;	//	Offset poz pobierania x 1mm
	stPickOffsetA									:	ST_LrParametr;	//	Offset poz pobierania x 1 stopeń
	stPickOffsetB									:	ST_LrParametr;	//	Offset poz pobierania x 1 stopeń
	stPickOffsetC									:	ST_LrParametr;	//	Offset poz pobierania x 1 stopeń
	                                                                      	
	stPickAccelecation								:	ST_UdiParametr;	//	Acc in % [1..100]
	stPickDecceleration								:	ST_UdiParametr;	//	Dec in % [1..100]
	stPickOverride									:	ST_UdiParametr;	//	Override in % [1..100]
	stPickColisionDetect							:	ST_UdiParametr; //	Col awoid in %[1..100]
	stPickGripperDelayTime							:	ST_UdiParametr;	//	Czas dojazdu   ms
	stSuckingTimeOn									:	ST_UdiParametr;	//	Czas posysania ms
	stSuckingTimeOff								:	ST_UdiParametr; //	Czas posysania ms
                                                                          	
	stPlaceOffsetX									:	ST_LrParametr;	//	Offset poz odkladania 2 x 1mm
	stPlaceOffsetY									:	ST_LrParametr;	//	Offset poz odkladania 2 x 1mm
	stPlaceOffsetZ									:	ST_LrParametr;	//	Offset poz odkladania 2 x 1mm
	stPlaceOffsetA									:	ST_LrParametr;	//	Offset poz odkladania 2 x 1 stopeń
	stPlaceOffsetB									:	ST_LrParametr;	//	Offset poz odkladania 2 x 1 stopeń
	stPlaceOffsetC									:	ST_LrParametr;	//	Offset poz odkladania 2 x 1 stopeń
                                                                          	
	stPlaceAccelecation								:	ST_UdiParametr;	//	Acc in % [1..100]
	stPlaceDecceleration							:	ST_UdiParametr;	//	Dec in % [1..100]
	stPlaceOverride									:	ST_UdiParametr;	//	Override in % [1..100]
	stPlaceColisionDetect							:	ST_UdiParametr; //	Col awoid in %[1..100]
	stRezerwa1										:	ST_UdiParametr;	//	
	stRezerwa2										:	ST_UdiParametr; //	
	stRezerwa3										:	ST_UdiParametr;	//	
	stGripperTimeClose								:	ST_UdiParametr;	//	Czas skłądania chwytaka
	stGripperTimeOpen								:	ST_UdiParametr;	//	Czas otwierania chwytaka
	                                                                      	
	stPickPreX										:	ST_LrParametr;	//	Odsuniecie przed pozycją pobierania w osi X      
	stPickPreY										:	ST_LrParametr;	//	Odsuniecie przed pozycją pobierania w osi Y      	
	stPickPreZ										:	ST_LrParametr;	//	Odsuniecie przed pozycją pobierania w osi Z      
	stPickAfterX									:	ST_LrParametr;  //	Odsuniecie po pobraniu w osi X                   
	stPickAfterY		                            :	ST_LrParametr;  //	Odsuniecie po pobraniu w osi Y                   
	stPickAfterZ		                            :	ST_LrParametr;  //	Odsuniecie po pobraniu w osi Z                   
	stPlacePreX										:	ST_LrParametr;  //	Odsuniecie przed pozycją odłożenia w osi X       
	stPlacePreY		                                :	ST_LrParametr;  //	Odsuniecie przed pozycją odłożenia w osi Y       
	stPlacePreZ		                                :	ST_LrParametr;  //	Odsuniecie przed pozycją odłożenia w osi Z       
	stPlaceAfterX		                            :	ST_LrParametr;  //	Odsuniecie po odłożenia w osi X                  
	stPlaceAfterY		                            :	ST_LrParametr;  //	Odsuniecie po odłożenia w osi Y                  
	stPlaceAfterZ		                            :	ST_LrParametr;  //	Odsuniecie po odłożenia w osi Z                  
	stBoxPickHeight									:	ST_LrParametr;       
	stBoxWingDown	  	                            :	ST_LrParametr;  //	Dolna długość krawędzi skrzydła kartonu          
	stCurveMotionPositionZ	  	                    :	ST_LrParametr;  //	Wysokość osłon dla dokładnego wkładania
	stCurveDistanceX	                            :	ST_LrParametr;  //	Offset pozycji najeżdzania na balchę prowadzącą X
	stCurveDistanceY								:	ST_LrParametr;  //	Offset pozycji najeżdzania na balchę prowadzącą Y
	stCurveDistanceZ	                            :	ST_LrParametr;  //	Offset pozycji najeżdzania na balchę prowadzącą Z
	stCurveMotionAngleA								:	ST_LrParametr;  //	Kąt zaokrąglenia włozenia kartonu A
	stCurveMotionAngleB                             :	ST_LrParametr;  //	Kąt zaokrąglenia włozenia kartonu B

END_STRUCT
END_TYPE

// ---- POUs/Recipes/NewRecipes/RecipeParts/ST_DownTransporterRecipe.TcDUT
TYPE ST_DownTransporterRecipe :
STRUCT
	wsCaption											:	WSTRING;	//Nazwa stacji	
	stTransporterVelocity								:	ST_UdiParametr;
END_STRUCT
END_TYPE

// ---- POUs/Recipes/NewRecipes/RecipeParts/ST_DymmyStationRecipe.TcDUT
TYPE ST_DymmyStationRecipe :
STRUCT
	wsCaption											:	WSTRING;	//Nazwa stacji	
END_STRUCT
END_TYPE

// ---- POUs/Recipes/NewRecipes/RecipeParts/ST_ExtMachineRecipe.TcDUT
TYPE ST_ExtMachineRecipe :
STRUCT
	wsCaption											:	WSTRING;	//Nazwa stacji	
	stUseComunication									:	ST_BoolParametr;
END_STRUCT
END_TYPE

// ---- POUs/Recipes/NewRecipes/RecipeParts/ST_InBoxControlRecipe.TcDUT
TYPE ST_InBoxControlRecipe :
STRUCT
	wsCaption											:	WSTRING;	//Nazwa stacji	
	stControlMode										:	ST_UdiParametr;
	stRejectDelay										:	ST_UdiParametr;
END_STRUCT
END_TYPE

// ---- POUs/Recipes/NewRecipes/RecipeParts/ST_InTransporterRecipe.TcDUT
TYPE ST_InTransporterRecipe :
STRUCT
	wsCaption											:	WSTRING;	//Nazwa stacji	
	stTransporterVelocity								:	ST_UdiParametr;
	stInTransporterWidth								: 	ST_LrParametr;	
	stInTransporterLength								: 	ST_LrParametr;	
END_STRUCT
END_TYPE

// ---- POUs/Recipes/NewRecipes/RecipeParts/ST_LeftRightCloserValveRecipe.TcDUT
TYPE ST_LeftRightCloserValveRecipe :
STRUCT
	wsCaption											:	WSTRING;	//Nazwa stacji	
	stWidthOffset										:	ST_LrParametr;
END_STRUCT
END_TYPE

// ---- POUs/Recipes/NewRecipes/RecipeParts/ST_LiftedTableRecipe.TcDUT
TYPE ST_LiftedTableRecipe :
STRUCT
	wsCaption											:	WSTRING;	//Nazwa stacji	
END_STRUCT
END_TYPE

// ---- POUs/Recipes/NewRecipes/RecipeParts/ST_LRTransporterRecipe.TcDUT
TYPE ST_LRTransporterRecipe :
STRUCT
	wsCaption											:	WSTRING;	//Nazwa stacji	
	stPositionL											:	ST_LrParametr;
	stPositionR											:	ST_LrParametr;
	stTransporterVelocityL								:	ST_UdiParametr;
	stTransporterVelocityR								:	ST_UdiParametr;
END_STRUCT
END_TYPE

// ---- POUs/Recipes/NewRecipes/RecipeParts/ST_MacroBoxFeedingProcessRecipe.TcDUT
TYPE ST_MacroBoxFeedingProcessRecipe :
STRUCT
	wsCaption											:	WSTRING;	//Nazwa stacji	
	stAnglePlace										:	ST_BoolParametr;
	stMaxTryCount										:	ST_UdiParametr;
	
	stSafeZposForMover									:	ST_LrParametr;
END_STRUCT
END_TYPE

// ---- POUs/Recipes/NewRecipes/RecipeParts/ST_MacroBoxingProcessRecipe.TcDUT
TYPE ST_MacroBoxingProcessRecipe :
STRUCT
	wsCaption											:	WSTRING;	//Nazwa stacji	
	
(*001*)	stReadyPos										:	ST_LrParametr;

(*002*)	stEndPos										:	ST_LrParametr;
(*003*)	stStartMoveTableDuringGoEndPos					:	ST_LrParametr; //To mid pos
	
(*005*)	stClosePos										:	ST_LrParametr;
(*006*)	stStartMoveTableDuringGoClosePos				:	ST_LrParametr;
	
(*007*)	stMovePos										:	ST_LrParametr;
	
(*008*)	stBoxPickPos									:	ST_LrParametr;	
	
(*009*)	stStartMoveTableDuringGoMovePos					:	ST_LrParametr; //To mid pos											:	ST_LrParametr;

(*010*)	stSafePosForProductRobot						:	ST_LrParametr;

(*011*)	stValveOnPosition								:	ST_LrParametr;
(*008*)	stHidePos									:	ST_LrParametr;	
END_STRUCT
END_TYPE

// ---- POUs/Recipes/NewRecipes/RecipeParts/ST_MacroInProcessRecipe.TcDUT
TYPE ST_MacroInProcessRecipe :
STRUCT
	wsCaption											:	WSTRING;	//Nazwa stacji	
	stProductPuttingInTime								:	ST_UdiParametr;
	stProductQueryWaitTime								:	ST_UdiParametr;
	stFallRSensor										: 	ST_BoolParametr;
	stCapSensor											: 	ST_BoolParametr;	
	stFirstBottleValve									: 	ST_BoolParametr;
	stVacuumOffTimer									:	ST_UdiParametr;
	stVacuumOnTimer										:	ST_UdiParametr;
	stEndWaitTime										:	ST_UdiParametr;
END_STRUCT
END_TYPE

// ---- POUs/Recipes/NewRecipes/RecipeParts/ST_MacroMachineProcessRecipe.TcDUT
TYPE ST_MacroMachineProcessRecipe :
STRUCT
	wsCaption											:	WSTRING;	//Nazwa stacji	

END_STRUCT
END_TYPE

// ---- POUs/Recipes/NewRecipes/RecipeParts/ST_MacroProductProcessRecipe.TcDUT
TYPE ST_MacroProductProcessRecipe :
STRUCT
	wsCaption											:	WSTRING;	//Nazwa stacji	
	
	stGateUpDelay										:	ST_UdiParametr;
	stGateDownDelay										:	ST_UdiParametr;

	stUseBottleMode										:	ST_BoolParametr;
	stTableCoversEnable									:	ST_BoolParametr;

END_STRUCT
END_TYPE

// ---- POUs/Recipes/NewRecipes/RecipeParts/ST_MacroTransportRecipe.TcDUT
TYPE ST_MacroTransportRecipe :
	STRUCT
		wsCaption											:	WSTRING;	//Nazwa stacji	
		
		//Sendors tolerance
		udiSensor420timeOn									:	ST_UdiParametr;
		udiSensor420timeOff									:	ST_UdiParametr;
	
		udiSensor430timeOn									:	ST_UdiParametr;
		udiSensor430timeOff									:	ST_UdiParametr;
		
		udiSensor440timeOn									:	ST_UdiParametr;
		udiSensor440timeOff									:	ST_UdiParametr;
		
		//starting delay
		udiPb450StartDelay									:	ST_UdiParametr;
		udiTr460StartDelay									:	ST_UdiParametr;
		udiTr470StartDelay									:	ST_UdiParametr;
	
		//stopping delay
		udiPb450StopDelay									:	ST_UdiParametr;
		udiTr460StopDelay									:	ST_UdiParametr;
		udiTr470StopDelay									:	ST_UdiParametr;
		
		//jdnostka
		bUseProductBoxer									:	ST_BoolParametr;
		bIndependentWorkWay1								:	ST_BoolParametr;
		bIndependentWorkWay2								:	ST_BoolParametr;
	END_STRUCT
END_TYPE

// ---- POUs/Recipes/NewRecipes/RecipeParts/ST_MainProcessRecipe.TcDUT
TYPE ST_MainProcessRecipe :
STRUCT
	wsCaption											:	WSTRING(200);	//Nazwa stacji	
	stProductCountX										:	ST_UdiParametr;
	stProductCountY										:	ST_UdiParametr;
	stProductCountZ										:	ST_UdiParametr;
	stProductHeight										:	ST_LrParametr;
	stProductSizeX										:	ST_LrParametr;
	stProductSizeY										:	ST_LrParametr;
	stBoxSizeX											:	ST_LrParametr;
	stBoxSizeY											:	ST_LrParametr;	
	stBoxSizeZ											:	ST_LrParametr;	
	stUseBoxesTransporter								:	ST_BoolParametr;
	stProductType										:	ST_TextListParametr;
	sBitmapId											:	STRING := 'RecipeImages.rysunek 1BP_1';
END_STRUCT
END_TYPE

// ---- POUs/Recipes/NewRecipes/RecipeParts/ST_MainSystemRecipe.TcDUT
TYPE ST_MainSystemRecipe :
STRUCT
	wsCaption											:	WSTRING;	//Nazwa stacji	
	
END_STRUCT
END_TYPE

// ---- POUs/Recipes/NewRecipes/RecipeParts/ST_MoverPressValveRecipe.TcDUT
TYPE ST_MoverPressValveRecipe :
STRUCT
	wsCaption											:	WSTRING;	//Nazwa stacji	
END_STRUCT
END_TYPE

// ---- POUs/Recipes/NewRecipes/RecipeParts/ST_OutControlRecipe.TcDUT
TYPE ST_OutControlRecipe :
STRUCT
	wsCaption											:	WSTRING;	//Nazwa stacji	
	stUseControl										:	ST_BoolParametr;
	stMaxWaitSensorTime									: 	ST_UdiParametr;
	
END_STRUCT
END_TYPE

// ---- POUs/Recipes/NewRecipes/RecipeParts/ST_ProductBoxerRecipe.TcDUT
TYPE ST_ProductBoxerRecipe :
STRUCT
	wsCaption											:	WSTRING;	//Nazwa stacji	
	
END_STRUCT
END_TYPE

// ---- POUs/Recipes/NewRecipes/RecipeParts/ST_ProductRobotRecipe.TcDUT
TYPE ST_ProductRobotRecipe :
STRUCT
	wsCaption											:	WSTRING;	//	Nazwa stacji	
	                                                                      	
	stPickOffsetX									:	ST_LrParametr;	//	Offset poz pobierania x 1mm
	stPickOffsetY									:	ST_LrParametr;	//	Offset poz pobierania x 1mm
	stPickOffsetZ									:	ST_LrParametr;	//	Offset poz pobierania x 1mm
	stPickOffsetA									:	ST_LrParametr;	//	Offset poz pobierania x 1 stopeń
	stPickOffsetB									:	ST_LrParametr;	//	Offset poz pobierania x 1 stopeń
	stPickOffsetC									:	ST_LrParametr;	//	Offset poz pobierania x 1 stopeń
	                                                                      	
	stPickAccelecation								:	ST_UdiParametr;	//	Acc in % [1..100]
	stPickDecceleration								:	ST_UdiParametr;	//	Dec in % [1..100]
	stPickOverride									:	ST_UdiParametr;	//	Override in % [1..100]
	stPickColisionDetect							:	ST_UdiParametr; //	Col awoid in %[1..100]
	stPickGripperDelayTime							:	ST_UdiParametr;	//	Czas dojazdu   ms
	stSuckingTimeOn									:	ST_UdiParametr;	//	Czas posysania ms
	stSuckingTimeOff								:	ST_UdiParametr; //	Czas posysania ms
                                                                          	
	stPlaceOffsetX									:	ST_LrParametr;	//	Offset poz odkladania 2 x 1mm
	stPlaceOffsetY									:	ST_LrParametr;	//	Offset poz odkladania 2 x 1mm
	stPlaceOffsetZ									:	ST_LrParametr;	//	Offset poz odkladania 2 x 1mm
	stPlaceOffsetA									:	ST_LrParametr;	//	Offset poz odkladania 2 x 1 stopeń
	stPlaceOffsetB									:	ST_LrParametr;	//	Offset poz odkladania 2 x 1 stopeń
	stPlaceOffsetC									:	ST_LrParametr;	//	Offset poz odkladania 2 x 1 stopeń
                                                                          	
	stPlaceAccelecation								:	ST_UdiParametr;	//	Acc in % [1..100]
	stPlaceDecceleration							:	ST_UdiParametr;	//	Dec in % [1..100]
	stPlaceOverride									:	ST_UdiParametr;	//	Override in % [1..100]
	stPlaceColisionDetect							:	ST_UdiParametr; //	Col awoid in %[1..100]
	stRezerwa1										:	ST_UdiParametr;	//	
	stRezerwa2										:	ST_UdiParametr; //	
	stRezerwa3										:	ST_UdiParametr;	//	
	                                                                      	
	stDistanceTCP_X									:	ST_LrParametr; 	//	Parameter TCP narżędzia mm
	stDistanceTCP_Y									:	ST_LrParametr; 	//	Parameter TCP narżędzia mm
	stDistanceTCP_Z									:	ST_LrParametr; 	//	Parameter TCP narżędzia mm
	
	stPickPreX										:	ST_LrParametr;	//	Odsuniecie przed pozycją pobierania w osi X      
	stPickPreY										:	ST_LrParametr;	//	Odsuniecie przed pozycją pobierania w osi Y      	
	stPickPreZ										:	ST_LrParametr;	//	Odsuniecie przed pozycją pobierania w osi Z      
	stPickAfterX									:	ST_LrParametr;  //	Odsuniecie po pobraniu w osi X                   
	stPickAfterY		                            :	ST_LrParametr;  //	Odsuniecie po pobraniu w osi Y                   
	stPickAfterZ		                            :	ST_LrParametr;  //	Odsuniecie po pobraniu w osi Z                   
	stAfterPickSafeX								:	ST_LrParametr;	//	Pozycja zezwolenia wjazdu kolejenego rządu
	stPlacePreX										:	ST_LrParametr;  //	Odsuniecie przed pozycją odłożenia w osi X       
	stPlacePreY		                                :	ST_LrParametr;  //	Odsuniecie przed pozycją odłożenia w osi Y       
	stPlacePreZ		                                :	ST_LrParametr;  //	Odsuniecie przed pozycją odłożenia w osi Z       
	stPlaceAfterX		                            :	ST_LrParametr;  //	Odsuniecie po odłożenia w osi X                  
	stPlaceAfterY		                            :	ST_LrParametr;  //	Odsuniecie po odłożenia w osi Y                  
	stPlaceAfterZ		                            :	ST_LrParametr;  //	Odsuniecie po odłożenia w osi Z                  
	stProductHighOffsetZ	                        :	ST_LrParametr;  //	Wysokość produktu do ominięcia dla powrotu       
	stProductPickHeight								:	ST_LrParametr; 
END_STRUCT
END_TYPE

// ---- POUs/Recipes/NewRecipes/RecipeParts/ST_ProductTableCoverRecipe.TcDUT
TYPE ST_ProductTableCoverRecipe :
STRUCT
	wsCaption											:	WSTRING;	//Nazwa stacji	
END_STRUCT
END_TYPE

// ---- POUs/Recipes/NewRecipes/RecipeParts/ST_RejectBuforRecipe.TcDUT
TYPE ST_RejectBuforRecipe :
STRUCT
	wsCaption											:	WSTRING;	//Nazwa stacji	
	stUseCounter										:	ST_BoolParametr;
	stMaxCount											:	ST_UdiParametr;
	stWarningCount										:	ST_UdiParametr;
	
	stUseSensor											:	ST_BoolParametr;
	stSensorMaxTime										:	ST_UdiParametr;
	
END_STRUCT
END_TYPE

// ---- POUs/Recipes/NewRecipes/RecipeParts/ST_SpareElementsLockRecipe.TcDUT
TYPE ST_SpareElementsLockRecipe :
STRUCT
	wsCaption											:	WSTRING;	//Nazwa stacji	
END_STRUCT
END_TYPE

// ---- POUs/Recipes/NewRecipes/RecipeParts/ST_StandartGateRecipe.TcDUT
TYPE ST_StandartGateRecipe :
STRUCT
	wsCaption											:	WSTRING;	//Nazwa stacji	
END_STRUCT
END_TYPE

// ---- POUs/Recipes/NewRecipes/RecipeParts/ST_StepMoverRecipe.TcDUT
TYPE ST_StepMoverRecipe :
STRUCT
	wsCaption												:	WSTRING;	//Nazwa stacji
	
	stLowAcceleration										:	ST_LrParametr;
	stLowDeceleration										:	ST_LrParametr;
	stLowVelocity											:	ST_LrParametr;
	stLowJerk												:	ST_LrParametr;
	
	stHighAcceleration										:	ST_LrParametr;
	stHighDeceleration										:	ST_LrParametr;
	stHighVelocity											:	ST_LrParametr;
	stHighJerk												:	ST_LrParametr;
END_STRUCT
END_TYPE

// ---- POUs/Recipes/NewRecipes/ST_Recipe.TcDUT
TYPE ST_Recipe :
STRUCT
	stUBL												:	ST_Recipe_UBL_PARAM;
	stUCF												:	ST_Recipe_UCF_PARAM;
	stUBF												:	ST_Recipe_UBF_PARAM;

END_STRUCT
END_TYPE

// ---- POUs/Recipes/NewRecipes/ST_RecipeListItem.TcDUT
TYPE ST_RecipeListItem :
STRUCT
	bUsed												:	BOOL;	//Cell is not empty
	udiIndex											:	UDINT;	//Recipe index
	wsRecipeCaption										:	WSTRING(255);
	wsRecipeDescription									:	WSTRING(255);
	wsCreateDate										:	WSTRING(255);
END_STRUCT
END_TYPE

// ---- POUs/Recipes/NewRecipes/ST_Recipe_UBF_PARAM.TcDUT
TYPE ST_Recipe_UBF_PARAM :
STRUCT
	(******BottleSupplySorter********)	
(*******************************BottleSupplySorter Product Type**************************************************************************)	
	//Sorter butelek, typ produktu
	iBottleSorterProductTypeShow												:	ST_DIParametrr;					// 		Typ produktu
	uiBottleSorterIndexShow														:	ST_DIParametrr;					// 		Index butelki 	
	                                                                   
(*******************************BottleSupplySorterHopperTransporter**************************************************************************)	
	//Sorter butelek, transporter zasobnika
	bBottleSorterHopperTransporterEnableShow									:	ST_BoolParametr;					//  	Aktywacja
	iBottleSorterHopperConveyorRunningSpeedSVShow								:	ST_DIParametrr;	//:= 5;			// 		Prędkość | [%] (1-100)
	iBottleSorterHopperConveyorEmptyingSpeedSVShow								:	ST_DIParametrr;	//:= 7;			// 		Prędkość, opróżnianie	| [%] (1-100)
	iBottleSorterDistanceToFindElementOnTransferConveyorLimitRunningSVShow		:	ST_DIParametrr;	//:= 610; 		// 		Odległość do butelek | [mm] (10-10_000)                                  		
	iBottleSorterDistanceToFindElementOnTransferConveyorLimitEmptyingSVShow		:	ST_DIParametrr;	//:= 500; 		// 		Odległość do butelek - opróżnianie | [mm] (10-10_000)                                       		

(*******************************BottleSupplySorterTransferTransporter**************************************************************************)
	//Sorter butelek, transporter transferowy	
	bBottleSorterTransferTransporterEnableShow									:	ST_BoolParametr;					// 		Aktywacja
	iBottleSorterTransferConveyorRunningSpeedSVShow								:	ST_DIParametrr;	//:= 5;			// 		Prędkość | [%] (1-100)	
	iBottleSorterTransferConveyorEmptyingSpeedSVShow							:	ST_DIParametrr;	//:= 7;			// 		Prędkość, opróżnianie | [%] (1-100)
	iBottleSorterDistanceToFindElementOnSupplyConveyorDownstairsLimitSVShow		:	ST_DIParametrr;	//:= 600;			// 		Odległość do butelek - stop zasypu | [mm] (10-10_000)
                                                                               
(*******************************BottleSupplySorterSupplyTransporter**************************************************************************)	
	//Sorter butelek, transporter zasypowy
	bBottleSorterSupplyTransporterEnableShow									:	ST_BoolParametr;					// [H] 	Aktywacja
	uiBottleSorterSupplyTransporterRunningSpeedSVShow							:	ST_UdiParametr;		//:= 1_000;		// 		Prędkość | [obr/min] (10-10_000)	
	uiBottleSorterSupplyTransporterEmptingSpeedSVShow							:	ST_UdiParametr;		//:= 1_000;		// 		Prędkość, opróżnianie | [obr/min] (10-10_000)                                                                   
	lrBottleSorterModuloMoveOffsetSVShow										:   ST_LrParametr;				// 		Kat sprawdzania | [°] (1-360)	                                                                            
	//Logika zasypu - warunek pierwszy	                                                            
	iBottleSorterSensorsCountFirstConditionSVShow								:	ST_DIParametrr;					// 		Limit butelek
	iBottleSorterSupplyTimeFirstConditionSVShow									:	ST_DIParametrr;					// 		Czas zasypu | [ms] (10-10_000)                                                                                                    		
	//Logika zasypu - warunek drugi	 	                                                                                       		
	iBottleSorterSensorsCountSecondConditionMinSVShow							:	ST_DIParametrr;					// 		Limit butelek, min
	iBottleSorterSensorsCountSecondConditionMaxSVShow							:	ST_DIParametrr;					// 		Limit butelek, max
	iBottleSorterSupplyTimeSecondConditionSVShow								:	ST_DIParametrr;					// 		Czas zasypu | [ms] (10-10_000)                                                                                                  		
	//Logika zasypu - warunek trzeci 	                                                                                       		
	iBottleSorterSensorsCountThirdConditionSVShow								:	ST_DIParametrr;					// 		Limit butelek
	iBottleSorterSupplyTimeThirdConditionSVShow									:	ST_DIParametrr;					// 		Czas zasypu | [ms] (10-10_000)
	                                                                            	
(*******************************BottleSupplySorterWheel**************************************************************************)	
	//Sorter butelek, Stól
	bBottleSorterWeelEnableShow													:	ST_BoolParametr;					// [H]	Aktywacja
	lrBottleSorterWheelSpeedSVShow												:   ST_LrParametr; //:= 20;			// 		Prędkość | [obr/min] (5-100)	            
	lrBottleSorterWheelEmptyingSpeedSVShow										:   ST_LrParametr; //:= 30;			// 		Prędkość, opróżnianie | [obr/min] (5-100)	
		
(*******************************BottleSupplySorterBrush**************************************************************************)		
	//Sorter butelek, szczotka
	bBottleSorterBrushEnableShow												:	ST_BoolParametr;					//		Aktywacja
	lrBottleSorterBrushHeightPositionSVShow										:   ST_LrParametr; // := 71;			// 		Wysokosc | [mm] (10-200)	
	iBottleSorterBrushRunningSpeedSVShow										:	ST_DIParametrr; 		 			// 		Prędkość | [%] (1-100)	            
	iBottleSorterBrushEmptyingSpeedSVShow										:	ST_DIParametrr; 		 			// 		Prędkość, opróżnianie | [%] (1-100)                                                              		         	
	
(*********************************BottleSupplyRobot*******************************************************************)

	//Sorter butelek, robot
	bBottleSorterRobotEnableShow												:	ST_BoolParametr;					// 		Aktywacja     
	nBottleSorterRobotRecipeId													:	ST_UdiParametr;					//		Nr receptury                                                                   
	//Czasy przyssania i oddmuchu                                                                                                                              
	lrBottleSorterRemainingTimeToSuctionShow             						:   ST_LrParametr;				// 		Wyprzedzenie przyssania | [ms] (0-200)
	lrBottleSorterSuckerSuctionTimeShow											:   ST_LrParametr;				// 		Czas przyssania	| [ms] (10-1000)
    lrBottleSorterRemainingTimeToRejectShow             						:   ST_LrParametr;				// 		Wuprzedzenie oddmuchu | [ms] (0-200)
	lrBottleSorterEjectorPulseShow                                       		:   ST_LrParametr;				// 		Czas oddmuchu	| [ms] (10-1000)			                                                                                                    		                                                                                                        		
	//Pkt. poboru i dokładania                                                                                 		                                                                                                          		
	lrBottleSorterZPickAboveTheBottleSVShow										:   ST_LrParametr;				// 		Wysokość pobierania butelki
	lrBottleSorterZPickMoveSVShow												:   ST_LrParametr;				// 		Odległość zjazdu w dół łapanie butelki 	                                                                                               	   		                                                                                     		
	lrBottleSorterSafetyHeightSVShow											:   ST_LrParametr;	//:= 150;  		// 		Wysokość obracania chwytaka | [mm] (0-1000)

(*********************************BottleReciever*******************************************************************)

	//Sorter butelek, robot
	bBottleSorterRecieverEnableShow												:	ST_BoolParametr;					// 		Aktywacja   
	bBottleSorterRecieverSlot1EnableShow										:	ST_BoolParametr;					// 		Aktywacja  
	bBottleSorterRecieverSlot2EnableShow										:	ST_BoolParametr;				// 		Aktywacja  
	bBottleSorterRecieverSlot3EnableShow										:	ST_BoolParametr;					// 		Aktywacja  
	lrBottleSorterRecieverHeightPositionSVShow									:   ST_LrParametr;				// 		Wysokosc | [mm] (10-200)	

END_STRUCT
END_TYPE

// ---- POUs/Recipes/NewRecipes/ST_Recipe_UBL_PARAM.TcDUT
TYPE ST_Recipe_UBL_PARAM :
STRUCT
sRecipeNameShow										:WSTRING;									// Nazwa 
sRecipeDescriptionShow								:WSTRING(1000);			                    // Nazwa 
                                                                                                
sRecipeIndexShow									:STRING;				                    // Indeks 
nRecipeIndexShow									:	ST_DIParametrr;						    // Indeks 
                                                                                                
//Parametry opakowania                                                                          
iPackageCapTypeShow									:	ST_DIParametrr;						    // Typ nasadki
iPackageCapDiameterShow								:	ST_DIParametrr;					        // Średnica nasadki
                                                                                                
//[H] Praca w trybie wybuchowym                                                                 
bExEnableShow										:	ST_BoolParametr;					    // [H] Tryb EX
                                                                                                
// Podajnik butelek  	                                                                        
bBottleFeederEnableShow								:	ST_BoolParametr;   				        // Aktywacja
iBottleFeederTurntableVelocitySVShow				:	ST_UdiParametr;					        // Prędkość stołu
iBottleFeederBottleSensorDelayShow					:	ST_DIParametrr;					        // Opóźnienie wjazdu butelki
iBottleFeederFormGateDelayShow						:	ST_DIParametrr;						    // Czas otwarcia szlabanu formatek
iBottleFeederAllowFormDelayShow						:	ST_DIParametrr;					        // Czas po którym formatka zostaje wypuszczona bez butelki
                                                                                                
// Podajnik opakowań	                                                                        
bPucksInserterEnableShow							:	ST_BoolParametr;   				        // Aktywacja
iPucksInserterTurntableVelocitySVShow				:	ST_UdiParametr;					        // Prędkość stołu
iPucksInserterConveyorVelocitySVShow				:	ST_UdiParametr;					        // Prędkość transportera
iPucksInserterBottleSensorDelayShow					:	ST_DIParametrr;				            // Opóźnienie wjazdu butelki
iPucksInserterFormGateDelayShow						:	ST_DIParametrr;							// Czas otwarcia szlabanu formatek	
iPucksInserterAllowFormDelayShow					:	ST_DIParametrr;							// Czas po którym formatka zostaje wypuszczona bez butelki	
lrPucksInserterWheelOffsetShow						:   ST_LrParametr;					        // Offset karuzeli +-10 st.
lrPucksInserterWheelAccelerationShow				:   ST_LrParametr;					        // Przyspieszenie 
lrPucksInserterWheelVelocityShow					:   ST_LrParametr;				            // Prędkość 
lrPucksInserterHammerHeightSVShow					:   ST_LrParametr;				            // Zadana wysokość
                                                                                                
//Sorter butelek                                                                                
//Parametry receptur z innego sterownika                                                        
                                                                                                
//[H] Parametry szlabanów                                                                       
bGateBeforeDispencersEnableShow						:	ST_BoolParametr;					    // [H] Aktywacja
nGateBeforeDispencersTimeFormInsertingShow			:   ST_LrParametr;					        // [H] Czas wyjazdu formatki	
bGateAfterWeightEnableShow							:	ST_BoolParametr;					    // [H] Aktywacja
nGateAfterWeightTimeFormInsertingShow				:   ST_LrParametr;					        // [H] Czas wyjazdu formatki
bGateRobotEnableShow								:	ST_BoolParametr;					    // [H] Aktywacja
nGateRobotTimeFormInsertingShow						:   ST_LrParametr;					        // [H] Czas przejazdu formatki
                                                                                                
//Przeciaganie formatek pod dozownikami	lewe                                                    
bFormsDragingLeftEnableShow							:	ST_BoolParametr;					    // Aktywacja
lrFormsDragingLeftVelocityShow						:   ST_LrParametr;					        // Prędkość [mm/s] (100-1000)
lrFormsDragingLeftAccelerationShow					:   ST_LrParametr;					        // Przyspieszenie [mm/s2] (100-10000)
lrFormsDragingLeftDecelerationShow					:   ST_LrParametr;					        // Hamowanie [mm/s2] (100-10000)
//Przeciaganie formatek pod dozownikami	prawe	                                                
bFormsDragingRightEnableShow						:	ST_BoolParametr;					    // Aktywacja
lrFormsDragingRightVelocityShow						:   ST_LrParametr;					        // Prędkość [mm/s] (100-1000)   
lrFormsDragingRightAccelerationShow					:   ST_LrParametr;				            // Przyspieszenie [mm/s2] (100-1
lrFormsDragingRightDecelerationShow					:   ST_LrParametr;				            // Hamowanie [mm/s2] (100-10000)
                                                                                                
//Dozowniki                                                                                     
bDosingTwoPhasesShow								:	ST_BoolParametr;					    // Dozowanie dwu-fazowe
lrDispencersLifterReadyPositionShow					:   ST_LrParametr;					        // Pozycja gototości 
uiDispencerStartDosingDelayShow						:	ST_UdiParametr;					        // Zwłoka rozpoczęcia dozowania
bDispencer1EnableShow								:	ST_BoolParametr; 					    // Aktywacja dozownika 1                                                        			
bDispencer2EnableShow								:	ST_BoolParametr;					    // Aktywacja dozownika 2 
bDispencer3EnableShow								:	ST_BoolParametr; 					    // Aktywacja dozownika 3  
bDispencer4EnableShow								:	ST_BoolParametr;					    // Aktywacja dozownika 4  
                                                                                                
